(*
  :return: CamReady 
*)
METHOD GetCamStatus : BOOL
VAR_OUTPUT
  bConnectionOK  : BOOL;    // Camera connected
  bTeachOk       : BOOL;    // Teach successful
  nTeachedPoints : UDINT;   // Teached points for this job
  nScannedPoints : UDINT;   // Scanned points on current sheet  
  bCamStarted    : BOOL;    // Camera trigger is active, cam started
  bCamDone       : BOOL;    // Camera finished on CT
  bErrors        : ARRAY[1..GVL_Camera.nC_NbCamErrors] OF BOOL;  // generic error flag list
END_VAR
bConnectionOK  := NOT bConnectionErr OR bSimulate;
bTeachOk       := _bTeachOk OR bSimulate;
nTeachedPoints := nNbMarksTeach;
nScannedPoints := nNbMarksScanned;
bCamStarted    := _bCamTriggerStarted;
// camera finished
IF nNbVersion = cProtoVersion_110 THEN
  // Done: Trigger released and last sector was received
  bCamDone       := _bCamTriggerDone AND ((nSector >= nNbSectorTeach) OR (nSector = SINT_TO_DINT(-1)));
ELSE
  // Done: Trigger released and same all teached points are scanned // NOTE: this will not work if not all marks are detected by camera
  bCamDone       := _bCamTriggerDone AND (nScannedPoints>=nTeachedPoints);
END_IF
GetCamStatus := bConnectionOK AND bTeachOk;   // camera ready
END_METHOD

(*
  get array index to point ID in stored point table
  :returns: TRUE if found, FALSE else
*)
METHOD getPointIndex : BOOL
VAR_INPUT
  nId : UDINT;
END_VAR
VAR_OUTPUT
  nIndex : UDINT;
END_VAR
VAR
  nResultIdx : DINT;
END_VAR
// search corresponding point in table (search for same mark ID)

nResultIdx := binarySearch(1, TO_DINT(nNbMarksTeach), TO_DINT(nId));
IF nResultIdx = -1 THEN
  LogWarning(F_Concat3('Point with Id: ', TO_STRING(nId) , ' not found in saved teach points'));
  nIndex := 1;
  RETURN;
END_IF

nIndex := TO_UDINT(nResultIdx);
getPointIndex := TRUE;
END_METHOD

METHOD INTERNAL getSimCamPoint : ST_DeformationPointAccurate
VAR_INPUT
  fXMin : LREAL := 0.0;
	fXMax : LREAL := 0.0;
	fYMin : LREAL := 0.0;
	fYMax : LREAL := 0.0;
	
	fOffsetMin : LREAL := 0.0;
	fOffsetMax : LREAL := 0.0;
END_VAR
VAR_OUTPUT
  sO_CamPoint : ST_DeformationPointAccurate;
END_VAR
VAR_INST
  fbRand : DRAND;
END_VAR
fbRand();
sO_CamPoint.x_ref := (fXMin + (fXMax - fXMin));
fbRand();
sO_CamPoint.y_ref := (fYMin + (fYMax - fYMin));

fbRand();
sO_CamPoint.dx := (fOffsetMin + (fOffsetMax - fOffsetMin) * fbRand.Num);
fbRand();
sO_CamPoint.dy := (fOffsetMin + (fOffsetMax - fOffsetMin) * fbRand.Num);

sO_CamPoint.valid := _bSimCamPointValid;
getSimCamPoint := sO_CamPoint;
END_METHOD

METHOD InitLineCamera
VAR_INPUT
  nPrintUnitResolution         : UDINT;    (*printhead pixel resolution [dpi]*)
  nPrintUnitSubPx              : UDINT;    (*print unit subPixel resolution [SubPx]*)
  nPrintUnitWidth              : UDINT;    (*print unit width in [px]*)
  iCameraTrigger               : I_CameraTrigger;
END_VAR
_fCameraWidthNormal     := FC_CONV_SUBPX_TO_M( _nCameraWidth
                                             , LREAL_TO_UDINT(cCameraResolution)
                                             , 1);
_nPrintUnitWidthNormal  := nPrintUnitWidth;
_fPrintUnitCalTemp      := fC_PhPixelDistRefTemp;   // reference temperate for real pixel spacing of ph
_fPrintUnitWidthTC      := (nPrintUnitWidth * fC_PhPixelDistFactorAtRefTemp) / 1000;  // caluclate print unit with at calibration temperature [m]

SUPER^.Init( nPrintUnitResolution:=nPrintUnitResolution
           , nPrintUnitSubPx:=nPrintUnitSubPx
           , iCameraTrigger := iCameraTrigger
           , bUseCameraTrigger:=TRUE
           , bUseCameraTriggerFeedback:=TRUE);
END_METHOD

METHOD InitSimulation : BOOL
VAR_INPUT
  aCamSimScriptPath : T_MaxString;
END_VAR
_aCamSimScriptPath := aCamSimScriptPath;
END_METHOD

METHOD mJobStart : BOOL
// re-calculate teach points with previous received 'T' telegram 
//  handles case: teach telegram arrived before JobStart
IF sModus = 'T' THEN calcTeachPoints(); END_IF
END_METHOD

(*
  Tcpip client rx message callback. 
  Called by FB_TcpMsgNotifier, registered with 'registerTcpIpClient()' before.
*)
METHOD rx_callback
VAR_INPUT
  sMessage : CalmarCompTcpIp.ST_TcpMsg;    // rx message
END_VAR
VAR
  sAnalyzeLastMessage    : STRING(GVL_TcpIp.TCP_RXDATA_SIZE);          // telegram string for analysis
  sTmpCamPoint           : ST_CameraPoint;
  
  nCounter               : UDINT;
  bOk, bEnd              : BOOL;

END_VAR
// basic message handling
SUPER^.rx_callback(sMessage := sMessage);
// debug print
IF _bVerbose THEN LogLvl(Lvl:=E_LogSeverity.Debug,Msg:=F_Concat4('Rx Sz: ', TO_STRING(nLastMessageSz), ' Msg:', sLastMessage)); END_IF

// check parameter (avoids crash)
IF _fPrintUnitWidthTC = 0 THEN LogError('rx_callback: Invalid configuration, review persistences and config values!'); RETURN; END_IF

// copy for parsing
sAnalyzeLastMessage := sLastMessage;      

REPEAT
  (*--- check message type ---*)
  // -- Is it a test message?
  IF rx_TestMsg(pMessage:=ADR(sLastMessage)) THEN       (*Test message*)
    RETURN;   // test message, ignore rest of parsing
   
  // -- Is it a error message ?
  ELSIF rx_ErrorMsg(pMessage:=ADR(sLastMessage)) THEN   (*Error message*)
    RETURN;   // error message, ignore rest of parsing
  
  // -- Is it a position message ('T' Teach or 'A' Auswertung)
  ELSIF rx_ParseHeader( pAnalyzeLastMessage := ADR(sAnalyzeLastMessage)
                      , nNbVersion      => nNbVersion          (*version*)
                      , sModus          => sModus              (*modus*)
                      , nNbMarks        => nNbMarks            (*number of marks*)
                      , nSector         => nSector)            (*sector*)
    THEN
     // got a position message, do not exit and do rest of parsing below
     // >>> DO parsing below 
     ;
    
  // -- unknown message
  ELSE
    IF _bVerbose THEN LogLvl(Lvl:=E_LogSeverity.Debug, Msg:=F_Concat2('unknown rx message (ignore): ', sLastMessage)); END_IF
    RETURN;
  END_IF
  
  
  (*--- Handle position telegram ---*)
  IF (sModus  = 'T') THEN 
    (*-- 'T' Teach message *)
    nNbMarksTeach   := 0;
    nNbMarksScanned := 0;
    nNbSectorTeach  := nSector;  (*Total number or sectors are send with teach message.*)
    sTeach          := sAnalyzeLastMessage; // display on visu
    
    IF _bVerbose THEN LogLvl(Lvl:=E_LogSeverity.Debug, Msg:='receive T telegram, erase cam/teach points list'); END_IF    
    MEMSET(destAddr:=ADR(sTeachPoints),  fillByte:=0, n:=SIZEOF(sTeachPoints));   // eraase teach points list
    MEMSET(destAddr:=ADR(sCameraPoints), fillByte:=0, n:=SIZEOF(sCameraPoints));  // erase cam points list
    MEMSET(destAddr:=ADR(nNumPointsPerSectorA), fillByte:=0, n:=SIZEOF(nNumPointsPerSectorA));
    MEMSET(destAddr:=ADR(nNumPointsPerSectorT), fillByte:=0, n:=SIZEOF(nNumPointsPerSectorT));
  ELSE
    (*-- 'A' Auswertung message *)
    sMemLastMessage := sAnalyzeLastMessage; // display on visu
    
    IF nSector = TO_DINT(cIdxFirstSector) THEN  // erase campoint with first received sector
      MEMSET(destAddr:=ADR(sCameraPoints), fillByte:=0, n:=SIZEOF(sCameraPoints));  // erase cam points list
      IF _bVerbose THEN LogLvl(Lvl:=E_LogSeverity.Debug, Msg:=F_Concat2('received first A sector, erase cam points list.','')); END_IF
      
      _nTimeFrameIdx_CamMsg := 1;
    END_IF
  
    // debug timing rx A
    IF _nTimeFrameIdx_CamMsg <= nC_MaxRxTimingEntries THEN  // save message timestamp for debugging
      _tTimeFrames_CamMsg[_nTimeFrameIdx_CamMsg] := F_GetCurDcTaskTime64();     // save cam frame rx timestamp
      _tTimeFramesMs_CamMsg[_nTimeFrameIdx_CamMsg] := TO_LREAL((_tTimeFrames_CamMsg[_nTimeFrameIdx_CamMsg]-_tTimeTrigger)/EC_DCTIME_TICKSPERMSEC64);  // delta to trigger in ms
      IF _bVerbose THEN 
        // dbg log rx frames
        LogLvl(Lvl:=E_LogSeverity.Debug, Msg:=F_Concat4(
            F_Concat2('A-Frame: ', TO_STRING(_nTimeFrameIdx_CamMsg)),
            F_Concat2(' : ', TO_STRING(_nTimeFrameIdx_CamMsg)),
            F_Concat2(' after trig: ', TO_STRING(_tTimeFramesMs_CamMsg[_nTimeFrameIdx_CamMsg])),
            F_Concat2(' at: ', TO_STRING(_tTimeFrames_CamMsg[_nTimeFrameIdx_CamMsg]))
        ));
			END_IF
      _nTimeFrameIdx_CamMsg := _nTimeFrameIdx_CamMsg + 1;
    END_IF
    
  END_IF;
  
  
  (*Search for rx, ry, lx, ly, v, x and y*)
  FOR nCounter := 1 TO nNbMarks DO
    // get next point
    IF NOT rx_ParsePoint(pAnalyzeLastMessage:=ADR(sAnalyzeLastMessage), sCamResult=>sTmpCamPoint, bLast=>bEnd) THEN 
      // invalid point received
      LogWarning(F_Concat2(
        F_Concat3('invalid ', SEL(sModus='T', 'camera', 'teach'), ' point received, '),
        F_CamPoint_ToString(sPoint:=sTmpCamPoint)
      ));
    END_IF
    IF bEnd AND nCounter < nNbMarks THEN LogWarning(F_Concat4('Less marks received than indicated in header: ', TO_STRING(nCounter), '<', TO_STRING(nNbMarks))); END_IF
    
    IF (sModus  = 'T') THEN
      (*-- 'T' Teach message *)
      // save (convert with job start)
      saveTeachPoint(sCamPoint := sTmpCamPoint);
    ELSE
      (*-- 'A' Auswertung message *)
      // save & convert cam point
      stCamPoint := saveAuswertungPoint(sCamPoint:=sTmpCamPoint, bOK=>bOk);     
      // stream point (if valid)
      IF bOk THEN  //AND sTmpCamPoint.valid THEN
        IF _iCameraSink <> 0 THEN
          _iCameraSink.AddCamPoint(stCamPoint);
          IF _bVerbose THEN 
            LogLvl(Lvl:=E_LogSeverity.Debug, Msg:= F_Concat2('AddCamPoint: ', F_DeformationPointAcc_ToString(sPointAcc:=stCamPoint)));
          END_IF
        END_IF
      END_IF
    END_IF
  END_FOR
UNTIL FIND2(ADR(sAnalyzeLastMessage), ADR(cStartString)) = 0   (*Search for another start string*)
END_REPEAT

IF (sModus  = 'T') THEN calcTeachPoints(); END_IF  // calculate teach points if it was a teach

bMsgReceived := FALSE;
END_METHOD

METHOD PRIVATE rx_DeleteMsgPart
VAR_INPUT
  pAnalyzeLastMessage    : POINTER TO STRING(GVL_TcpIp.TCP_RXDATA_SIZE);  // telegram string for analysis
  nLen                   : UDINT;
  nPos                   : UDINT;
END_VAR
VAR
  sMessageDelete         : STRING(GVL_TcpIp.TCP_RXDATA_SIZE);             // telegram string for analysis
END_VAR
DELETE2( pSrcString := pAnalyzeLastMessage
       , pDstString := ADR(sMessageDelete)
       , nDstSize   := SIZEOF(sMessageDelete)
       , nLen       := nLen
       , nPos       := nPos);

pAnalyzeLastMessage^ := sMessageDelete;
END_METHOD

(*
  Parse for error message
  :return: TRUE if it was an error test telegram, FALSE if other.
*)
METHOD PRIVATE rx_ErrorMsg : BOOL
VAR_INPUT
  pMessage    : POINTER TO STRING(GVL_TcpIp.TCP_RXDATA_SIZE);   // tcp message string pointer 
END_VAR
VAR
  nFIdx : UDINT;    // string find index
  nFrmIdx : UDINT;
  tDiff : LREAL;
  sErrMsg : T_MaxString;
END_VAR
// parse message type
nFIdx := FIND2(pMessage, ADR(cErrorString));
IF nFIdx > 0 THEN  
  IF _bVerbose THEN LogLvl(Lvl:=E_LogSeverity.Debug, Msg:=F_Concat2('error: msg received: ', pMessage^)); END_IF

  // error telegram received
  DELETE2( pSrcString := pMessage
         , pDstString := ADR(sErrMsg)
         , nDstSize   := SIZEOF(sErrMsg)
         , nLen       := (nFIdx + INT_TO_UDINT(LEN(cErrorString)) - 1)
         , nPos       := 1);

  // strip other control characters
  FindAndDelete(pSrcString:=ADR(sErrMsg), pDstString:=ADR(sErrMsg), nDstSize:=SIZEOF(sErrMsg), pDeleteString:=ADR(cEndingString));
  
  // error message implement handling
  
  rx_ErrorMsg := TRUE;
ELSE
  ; // other telegram
END_IF
END_METHOD

(*
  Parse for position telegram header.
  :return: TRUE if valid position telegram, FALSE else
*)
METHOD PRIVATE rx_ParseHeader : BOOL
VAR_INPUT
  pAnalyzeLastMessage    : POINTER TO STRING(GVL_TcpIp.TCP_RXDATA_SIZE);  // telegram string for analysis
END_VAR
VAR_OUTPUT
  nNbVersion             : INT;                   (*(V) Version: protocol version, e.g. 100/110/...*)
  sModus                 : T_MaxString;           (*(M) Modus: 'T'/'A'*)
  nNbMarks               : UDINT;                 (*(A) Merkmale: number of Marks in Teach/Auswertung*)
  nSector                : DINT;                  (*(S) Sectors: Number of Sectors in 'T' / Sector index in 'A'*)
  //sMemLastMessage        : STRING(GVL_TcpIp.TCP_RXDATA_SIZE);  (*rx telegram string without header*)
END_VAR
VAR
  nFindIndex             : UDINT;
END_VAR
(*Search for start string*)
nFindIndex := FIND2(pAnalyzeLastMessage, ADR(cStartString));
IF nFindIndex = 0 THEN RETURN; END_IF

(*Search string found => remove string to evaluate rest of message*)
rx_DeleteMsgPart(pAnalyzeLastMessage := pAnalyzeLastMessage, nLen := (nFindIndex + INT_TO_UDINT(LEN(cStartString)) - 1) , nPos := 1);

(*Search for version number*)
nFindIndex := FIND2(pAnalyzeLastMessage, ADR(','));
IF nFindIndex > 0 THEN
  nNbVersion := STRING_TO_INT(LEFT(pAnalyzeLastMessage^, (UDINT_TO_INT(nFindIndex) - 1)));

  rx_DeleteMsgPart(pAnalyzeLastMessage := pAnalyzeLastMessage, nLen := nFindIndex , nPos := 1);
END_IF;

(*Search for modus (M)*)
nFindIndex := FIND2(pAnalyzeLastMessage, ADR(','));
IF nFindIndex > 0 THEN
  sModus := LEFT(pAnalyzeLastMessage^, (UDINT_TO_INT(nFindIndex) - 1));

  rx_DeleteMsgPart(pAnalyzeLastMessage := pAnalyzeLastMessage, nLen := nFindIndex , nPos := 1);
END_IF;

(*Search for number marks (A)*)
nFindIndex := FIND2(pAnalyzeLastMessage, ADR(','));
IF nFindIndex > 0 THEN
  nNbMarks := STRING_TO_UDINT(LEFT(pAnalyzeLastMessage^, (UDINT_TO_INT(nFindIndex) - 1)));
  IF nNbMarks > GVL_Camera.cMaxNbMarks THEN
    LogLvl(Lvl:=E_LogSeverity.Warning, Msg:=F_Concat4('Limit marks (', TO_STRING(nNbMarks),') to max=', TO_STRING(GVL_Camera.cMaxNbMarks)));
    nNbMarks := GVL_Camera.cMaxNbMarks;
  END_IF

  rx_DeleteMsgPart(pAnalyzeLastMessage := pAnalyzeLastMessage, nLen := nFindIndex , nPos := 1);
END_IF;

(*Search for sector of transmission (S)*)
nFindIndex := FIND2(pAnalyzeLastMessage, ADR(','));
IF nFindIndex > 0 THEN
  (*Last sector is indicated with '-1'*)
  nSector := STRING_TO_DINT(LEFT(pAnalyzeLastMessage^, (UDINT_TO_INT(nFindIndex) - 1)));

  rx_DeleteMsgPart(pAnalyzeLastMessage := pAnalyzeLastMessage, nLen := nFindIndex , nPos := 1);
ELSE
  // end of message detected
  nFindIndex := FIND2(pAnalyzeLastMessage, ADR(');'));
  IF nFindIndex > 0 THEN
    (*Last sector is indicated with '-1'*)
    nSector := STRING_TO_DINT(LEFT(pAnalyzeLastMessage^, (UDINT_TO_INT(nFindIndex) - 1)));
  
    rx_DeleteMsgPart(pAnalyzeLastMessage := pAnalyzeLastMessage, nLen := nFindIndex + 1, nPos := 1);
  END_IF;
END_IF;

rx_ParseHeader := TRUE;
END_METHOD

(*
  Parse a point entry from string.
  And removes this string part from pAnalyzeLastMessage.
  :return: TRUE if point is valid
*)
METHOD PRIVATE rx_ParsePoint : BOOL
VAR_INPUT
  pAnalyzeLastMessage    : POINTER TO STRING(GVL_TcpIp.TCP_RXDATA_SIZE);  // telegram string for analysis
END_VAR
VAR_OUTPUT
  sCamResult             : ST_CameraPoint;
  bLast                  : BOOL;
END_VAR
VAR
  nFindIndex             : UDINT;
END_VAR
(*Index of mark (T)*)
nFindIndex := FIND2(pAnalyzeLastMessage, ADR(','));
IF nFindIndex > 0 THEN
  sCamResult.id := STRING_TO_UDINT(LEFT(pAnalyzeLastMessage^, (UDINT_TO_INT(nFindIndex) - 1)));
  
  rx_DeleteMsgPart(pAnalyzeLastMessage := pAnalyzeLastMessage, nLen := nFindIndex , nPos := 1);
END_IF;

(*rx*)
nFindIndex := FIND2(pAnalyzeLastMessage, ADR(','));
IF nFindIndex > 0 THEN
  sCamResult.x_ref := STRING_TO_DINT(LEFT(pAnalyzeLastMessage^, (UDINT_TO_INT(nFindIndex) - 1)));

  IF    (sCamResult.x_ref < cCameraMinXY)
     OR (sCamResult.x_ref > cCameraMaxXY)
  THEN
    sCamResult.valid := FALSE;
  END_IF;

  rx_DeleteMsgPart(pAnalyzeLastMessage := pAnalyzeLastMessage, nLen := nFindIndex , nPos := 1);
ELSE
  sCamResult.valid := FALSE;
END_IF;
(*ry*)
nFindIndex := FIND2(pAnalyzeLastMessage, ADR(','));
IF nFindIndex > 0 THEN
  sCamResult.y_ref := STRING_TO_DINT(LEFT(pAnalyzeLastMessage^, (UDINT_TO_INT(nFindIndex) - 1)));

  IF    (sCamResult.y_ref < cCameraMinXY)
     OR (sCamResult.y_ref > cCameraMaxXY)
  THEN
    sCamResult.valid := FALSE;
  END_IF;

  rx_DeleteMsgPart(pAnalyzeLastMessage := pAnalyzeLastMessage, nLen := nFindIndex , nPos := 1);
ELSE
  sCamResult.valid := FALSE;
END_IF;

(*lx*)
nFindIndex := FIND2(pAnalyzeLastMessage, ADR(','));
IF nFindIndex > 0 THEN
  sCamResult.lx := STRING_TO_DINT(LEFT(pAnalyzeLastMessage^, (UDINT_TO_INT(nFindIndex) - 1)));

  IF    (sCamResult.lx < cCameraMinXY)
     OR (sCamResult.lx > cCameraMaxXY)
  THEN
    sCamResult.valid := FALSE;
  END_IF;

  rx_DeleteMsgPart(pAnalyzeLastMessage := pAnalyzeLastMessage, nLen := nFindIndex , nPos := 1);
ELSE
  sCamResult.valid := FALSE;
END_IF;
(*ly*)
nFindIndex := FIND2(pAnalyzeLastMessage, ADR(','));
IF nFindIndex > 0 THEN
  sCamResult.ly := STRING_TO_DINT(LEFT(pAnalyzeLastMessage^, (UDINT_TO_INT(nFindIndex) - 1)));

  IF    (sCamResult.ly < cCameraMinXY)
     OR (sCamResult.ly > cCameraMaxXY)
  THEN
    sCamResult.valid := FALSE;
  END_IF;

  rx_DeleteMsgPart(pAnalyzeLastMessage := pAnalyzeLastMessage, nLen := nFindIndex , nPos := 1);
ELSE
  sCamResult.valid := FALSE;
END_IF;

(*v*)
nFindIndex := FIND2(pAnalyzeLastMessage, ADR(','));
IF nFindIndex > 0 THEN
  IF STRING_TO_INT(LEFT(pAnalyzeLastMessage^, (UDINT_TO_INT(nFindIndex) - 1))) = 1 THEN
    sCamResult.valid := TRUE;
  ELSE
    sCamResult.valid := FALSE;
  END_IF;

  rx_DeleteMsgPart(pAnalyzeLastMessage := pAnalyzeLastMessage, nLen := nFindIndex , nPos := 1);
ELSE
  sCamResult.valid := FALSE;
END_IF;
(*x*)
nFindIndex := FIND2(pAnalyzeLastMessage, ADR(','));
IF nFindIndex > 0 THEN
  sCamResult.x := STRING_TO_DINT(LEFT(pAnalyzeLastMessage^, (UDINT_TO_INT(nFindIndex) - 1)));

  IF    (sCamResult.x < cCameraMinXY)
     OR (sCamResult.x > cCameraMaxXY)
  THEN
    sCamResult.valid := FALSE;
  END_IF;

  rx_DeleteMsgPart(pAnalyzeLastMessage := pAnalyzeLastMessage, nLen := nFindIndex , nPos := 1);
ELSE
  sCamResult.valid := FALSE;
END_IF;
(*y*)
nFindIndex := FIND2(pAnalyzeLastMessage, ADR(','));
IF (nFindIndex > 0) AND (nFindIndex <= 8) THEN  (*nFindIndex is > 8 if a second message is in the frame*)
  sCamResult.y := STRING_TO_DINT(LEFT(pAnalyzeLastMessage^, (UDINT_TO_INT(nFindIndex) - 1)));

  IF    (sCamResult.y < cCameraMinXY)
     OR (sCamResult.y > cCameraMaxXY)
  THEN
    sCamResult.valid := FALSE;
  END_IF;

  rx_DeleteMsgPart(pAnalyzeLastMessage := pAnalyzeLastMessage, nLen := nFindIndex , nPos := 1);
ELSE
  nFindIndex := FIND2(pAnalyzeLastMessage, ADR(');'));
  IF nFindIndex > 0 THEN
    sCamResult.y := STRING_TO_DINT(LEFT(pAnalyzeLastMessage^, (UDINT_TO_INT(nFindIndex) - 1)));
    bLast := TRUE;
    IF    (sCamResult.y < cCameraMinXY)
       OR (sCamResult.y > cCameraMaxXY)
    THEN
      sCamResult.valid := FALSE;
    END_IF;

    rx_DeleteMsgPart(pAnalyzeLastMessage := pAnalyzeLastMessage, nLen := nFindIndex + 1, nPos := 1);
  ELSE
    sCamResult.valid := FALSE;
  END_IF;
END_IF;

rx_ParsePoint := sCamResult.valid;
END_METHOD

(*
  Parse rx test telegrams.
  :return: TRUE if it was a known test telegram, FALSE if other.
*)
METHOD PRIVATE rx_TestMsg : BOOL
VAR_INPUT
  pMessage    : POINTER TO STRING(GVL_TcpIp.TCP_RXDATA_SIZE);   // tcp message string pointer 
END_VAR
VAR
  nFIdx : UDINT;    // string find index
  nFrmIdx : UDINT;
  tDiff : LREAL;
  sTestMsg : T_MaxString;
END_VAR
// rx timestamp
_tTimeRx := F_GetCurDcTaskTime64();

// parse message type
nFIdx := FIND2(pMessage, ADR(sQvTest_Header));
IF nFIdx > 0 THEN  
  IF _bVerbose THEN
    LogLvl(Lvl:=E_LogSeverity.Debug, Msg:=F_Concat2('test_rx: msg received: ', pMessage^));
  END_IF
  
  // test telegram received
  DELETE2( pSrcString := pMessage
         , pDstString := ADR(sTestMsg)
         , nDstSize   := SIZEOF(sTestMsg)
         , nLen       := (nFIdx + INT_TO_UDINT(LEN(sQvTest_Header)) - 1)
         , nPos       := 1);

  // strip QR start and end characters
  FindAndDeleteChar(pSrcString:=ADR(sTestMsg), pDstString:=ADR(sTestMsg), nDstSize:=SIZEOF(sTestMsg), sDeleteChar:='<');
  FindAndDeleteChar(pSrcString:=ADR(sTestMsg), pDstString:=ADR(sTestMsg), nDstSize:=SIZEOF(sTestMsg), sDeleteChar:=';');
  
  // Parse per test message type, e.g.  <QR_CI_1;
  // -- qv input frame timing test
  IF sQvTest_CI = LEFT(sTestMsg, LEN(sQvTest_CI)) THEN
    // strip header and test indication
    DELETE2( pSrcString := ADR(sTestMsg)
           , pDstString := ADR(sTestMsg)
           , nDstSize   := SIZEOF(sTestMsg)
           , nLen       := (1 + INT_TO_UDINT(LEN(sQvTest_CI)) - 1)
           , nPos       := 1);
    // frame number
    nFrmIdx := TO_UINT(sTestMsg);
    IF nFrmIdx <= nC_MaxRxTimingEntries THEN
      _tTimeFrames_TestMsg[nFrmIdx] := F_GetCurDcTaskTime64();     // save test input frame timestamp
      _tTimeFramesMs_TestMsg[nFrmIdx] := TO_LREAL((_tTimeFrames_TestMsg[nFrmIdx]-_tTimeTrigger)/EC_DCTIME_TICKSPERMSEC64);
    END_IF
    rx_TestMsg := TRUE;
    
  // -- qv loop time test frame response
  ELSIF sQvTest_Loop = LEFT(sTestMsg, LEN(sQvTest_Loop)) THEN
    tDiff := TO_LREAL((_tTimeRx - _tTimeTx) / EC_DCTIME_TICKSPERMSEC64); // calc time elapsed in [ms]
    _sTimeElapsed := F_Concat2(TO_STRING(tDiff),'ms');
    LogLvl(Lvl:=E_LogSeverity.Debug, Msg:=F_Concat2('rx_test: Loop time=', _sTimeElapsed));
    rx_TestMsg := TRUE;
  
  // -- unknown test message
  ELSE
    ;
	END_IF
ELSE
  ; // other telegram
END_IF
END_METHOD

METHOD PRIVATE saveAuswertungPoint : ST_DeformationPointAccurate
VAR_INPUT
  sCamPoint : ST_CameraPoint;
END_VAR
VAR_OUTPUT
  bOK : BOOL;   // conversion has been done correctly (ok as well if point is invalid!)
END_VAR
VAR
  nMarkIndex        : UDINT;
  fDistortionFactor : LREAL;                 (*distortion factor*)
END_VAR
(*convert and save Auswertungs point*)
IF NOT getPointIndex(nId:=sCamPoint.id, nIndex=>nMarkIndex) THEN
  LogError(F_Concat3('Auswertung point with Id: ', TO_STRING(sCamPoint.id), ' not found, ignore'));
  bOK := FALSE;
  RETURN;
END_IF

(*----- calculate print point position -----*)
(*Actual position of distinctive mark*)
(*NOTE: camera points have a different resolution! camera 300dpi * 16=4800dpi*)
IF sTeachPoints[nMarkIndex].x_teach_Print = 0 THEN 
  (*Fully automatic mode*)
  sTeachPoints[nMarkIndex].x_Print := FC_CONV_SUBPX_TO_M( sCamPoint.y
                                                          , LREAL_TO_UDINT(cCameraResolution)
                                                          , LREAL_TO_UDINT(cCameraResolutionSubpixel)) * 1000;  (*[m] => [mm]*)
ELSE
  (*Semi automatic mode*)
  sTeachPoints[nMarkIndex].x_Print :=     sTeachPoints[nMarkIndex].x_ref_Print
                                        + sTeachPoints[nMarkIndex].x_teach_Print
                                        - FC_CONV_SUBPX_TO_M( sCamPoint.y
                                                            , LREAL_TO_UDINT(cCameraResolution)
                                                            , LREAL_TO_UDINT(cCameraResolutionSubpixel)) * 1000;  (*[m] => [mm]*)
END_IF;
IF sTeachPoints[nMarkIndex].y_teach_Print = 0 THEN 
  (*Fully automatic mode*)
  sTeachPoints[nMarkIndex].y_Print :=   ((fPrintUnitWidthTAct/2 + fCameraWidthTC/2) * 1000)  (*[m] => [mm]*)
                                        - (  DINT_TO_LREAL(sCamPoint.x)
                                           / (fCameraRealResolution * cCameraResolutionSubpixel) * 25.4);  (*[mm]*)
ELSE
  (*Semi automatic mode*)
  sTeachPoints[nMarkIndex].y_Print :=     sTeachPoints[nMarkIndex].y_ref_Print
                                        + sTeachPoints[nMarkIndex].y_teach_Print
                                        - (  DINT_TO_LREAL(sCamPoint.x)
                                           / (fCameraRealResolution * cCameraResolutionSubpixel) * 25.4);  (*[mm]*)
END_IF;

// save cam point for visu
sCameraPoints[nMarkIndex] := sCamPoint;

(*----- create cam correction point -----*)
(*NOTE: correction will be rounded to [px]*)
saveAuswertungPoint.x_ref := F_MeterToSubPixelReal( sTeachPoints[nMarkIndex].x_ref_Print * 0.001      (*[mm] => [m]*)
                                     , UDINT_TO_LREAL(_nPrintUnitResolution));             (*Result should be in pixels*)                           
saveAuswertungPoint.y_ref := F_MeterToSubPixelReal( sTeachPoints[nMarkIndex].y_ref_Print * 0.001      (*[mm] => [m]*)
                                     , UDINT_TO_LREAL(_nPrintUnitResolution));             (*Result should be in pixels*)       
fCameraDelay := F_SubPixelToMeter(lPosSubPx:=_nCamStartPosDeviation, fResSubPx:=UDINT_TO_LREAL(_nPrintUnitResolution*_nPrintUnitSubPx));
saveAuswertungPoint.dx    := F_MeterToSubPixelReal( (sTeachPoints[nMarkIndex].x_ref_Print - sTeachPoints[nMarkIndex].x_Print) * 0.001  (*[mm] => [m]*)
                                     + fCameraDelay                                        (*apply camera trigger jitter*)
                                     , UDINT_TO_LREAL(_nPrintUnitResolution));             (*Result should be in pixels*)
                                     
(*Distortion due to expansion of print unit, calculate factor*)
fDistortionFactor := ((_fPrintUnitWidthTC / 2 * 1000) - sTeachPoints[nMarkIndex].y_ref_Print) / (_fPrintUnitWidthTC / 2 * 1000);
saveAuswertungPoint.dy := F_MeterToSubPixelReal( (  (sTeachPoints[nMarkIndex].y_ref_Print - sTeachPoints[nMarkIndex].y_Print)
                                     + fCameraAdjustmentY
                                     + ((fPrintUnitWidthDiff * 1000 / 2) * fDistortionFactor)   (*Distortion due to expansion of print unit*)
                                     + (fPrintUnitCenterOffsetTAct - fCameraCenterOffsetTAct)   (*Compensation due to unilateral expansion*)
                                    ) * 0.001  (*[mm] => [m]*)
                                  , UDINT_TO_LREAL(_nPrintUnitResolution));             (*Result should be in pixels*)
                                  
// not used entries
saveAuswertungPoint.index := 0; // optional: TO_DINT(sCamPoint.id);
saveAuswertungPoint.col := 0;
saveAuswertungPoint.row := 0;
saveAuswertungPoint.valid := sCamPoint.valid;
IF NOT sCamPoint.valid THEN     // erase spurious corrections on invalid points
  saveAuswertungPoint.dx := 0;
  saveAuswertungPoint.dy := 0;
END_IF
nNbMarksScanned := nNbMarksScanned + 1;
bOK := TRUE;
END_METHOD

METHOD PRIVATE saveTeachPoint
VAR_INPUT
  sCamPoint : ST_CameraPoint;
END_VAR
(*save teach point in table*)
// NOTE: mark ID unique and does not match the array index! 
IF nNbMarksTeach = GVL_Camera.cMaxNbMarks THEN 
  LogLvl(Lvl:=E_LogSeverity.Error, Msg:=F_Concat4('Too many marks received max. allowed: ', TO_STRING(GVL_Camera.cMaxNbMarks), ' ignore mark with id:', TO_STRING(sCamPoint.id)));
  RETURN;
END_IF

// save next teach mark
nNbMarksTeach := nNbMarksTeach + 1;
sCameraPoints[nNbMarksTeach] := sCamPoint;
END_METHOD

(*
  Set mode to camera.
  :return: TRUE if success
*)
METHOD setCameraMode : BOOL
VAR_INPUT
  eCameraMode : E_CameraMode;
END_VAR
IF eCameraMode = E_CameraMode.XYR OR   // supported modi
   eCameraMode = E_CameraMode.Auto OR
   eCameraMode = E_CameraMode.Live OR 
   eCameraMode = E_CameraMode.Trend THEN
   
  _eCameraMode := eCameraMode;  // set desired mode
  setCameraMode := TRUE;
ELSE
  LogError(F_Concat3('Camera mode=', TO_STRING(eCameraMode), ' not supported by camera'));
  _eCameraMode := E_CameraMode.NoCorrection;
END_IF
END_METHOD

METHOD SimEnter : BOOL
VAR_INST
  sSimMsg         : CalmarCompTcpIp.ST_TcpMsg;
  nFrameSize      : UDINT := 2048;
  nMarksPerFrame  : UDINT := 4;
END_VAR
IF NOT bSimEnable THEN RETURN; END_IF

IF    _nSimMode = 0 THEN
   //nNbMarksTeach := 4; // just somebigger than 2
   //nNbMarks := nNbMarksTeach;
ELSIF _nSimMode = 1 THEN
  // use external camera simulation script
  nFrameNr := 0;
ELSIF _nSimMode = 2 THEN
  // send directly some messages
  sSimMsg.stRemoteAddr.sAddr:='127.0.0.1';
  sSimMsg.stRemoteAddr.nPort:=3000;
  //v100 teach
  //rx_callback(sMessage:='<position(100,T,39,3,125,0,0,0,0,1,7184,7184,126,0,0,0,0,1,7184,26080,127,0,0,0,0,1,7184,35520,128,0,0,0,0,1,7184,54416,129,0,0,0,0,1,7168,73312,130,0,0,0,0,1,7184,82768,131,0,0,0,0,1,7184,101664,132,0,0,0,0,1,7184,120560,133,0,0,0,0,1,7184,139456,134,0,0,0,0,1,7184,148912,135,0,0,0,0,1,7184,167808,136,0,0,0,0,1,7168,186704,137,0,0,0,0,1,63872,7184,138,0,0,0,0,1,63872,26080,139,0,0,0,0,1,63872,35520,140,0,0,0,0,1,63872,54416,141,0,0,0,0,1,63872,73312,142,0,0,0,0,1,63872,82768,143,0,0,0,0,1,63872,101664,144,0,0,0,0,1,63872,120560,145,0,0,0,0,1,63872,139456,146,0,0,0,0,1,63872,148912,147,0,0,0,0,1,63872,167808,148,0,0,0,0,1,63872,186704,149,0,0,0,0,1,130016,7168,150,0,0,0,0,1,130016,26080,151,0,0,0,0,1,130016,35520,152,0,0,0,0,1,130016,54416,153,0,0,0,0,1,130016,73312,154,0,0,0,0,1,130016,82768,155,0,0,0,0,1,130016,101664,156,0,0,0,0,1,130016,120560,157,0,0,0,0,1,130016,139456,158,0,0,0,0,1,130016,148912,159,0,0,0,0,1,130016,167808,160,0,0,0,0,1,130016,186704,161,0,0,0,0,1,35520,7168,162,0,0,0,0,1,35520,5441);');
  //v110 teach
  sSimMsg.sMessage:= '<position(110,T,38,12,1,0,0,0,0,1,7184,7184,2,0,0,0,0,1,7184,26080,4,0,0,0,0,1,7184,35520,128,0,0,0,0,1,7184,54416,5,0,0,0,0,1,7168,73312,130,0,0,0,0,1,7184,82768,131,0,0,0,0,1,7184,101664,132,0,0,0,0,1,7184,120560,133,0,0,0,0,1,7184,139456,134,0,0,0,0,1,7184,148912,135,0,0,0,0,1,7184,167808,136,0,0,0,0,1,7168,186704,137,0,0,0,0,1,63872,7184,138,0,0,0,0,1,63872,26080,139,0,0,0,0,1,63872,35520,140,0,0,0,0,1,63872,54416,141,0,0,0,0,1,63872,73312,142,0,0,0,0,1,63872,82768,143,0,0,0,0,1,63872,101664,144,0,0,0,0,1,63872,120560,145,0,0,0,0,1,63872,139456,146,0,0,0,0,1,63872,148912,147,0,0,0,0,1,63872,167808,148,0,0,0,0,1,63872,186704,149,0,0,0,0,1,130016,7168,150,0,0,0,0,1,130016,26080,151,0,0,0,0,1,130016,35520,152,0,0,0,0,1,130016,54416,153,0,0,0,0,1,130016,73312,154,0,0,0,0,1,130016,82768,155,0,0,0,0,1,130016,101664,156,0,0,0,0,1,130016,120560,157,0,0,0,0,1,130016,139456,158,0,0,0,0,1,130016,148912,159,0,0,0,0,1,130016,167808,160,0,0,0,0,1,130016,186704,161,0,0,0,0,1,35520,7168,162,0,0,0,0,1,35520,5441);';
  //points 1 to 38
  //sSimMsg.sMessage:= '<position(110,T,38,12,1,0,0,0,0,1,7184,7184,2,0,0,0,0,1,7184,26080,3,0,0,0,0,1,7184,35520,4,0,0,0,0,1,7184,54416,5,0,0,0,0,1,7168,73312,6,0,0,0,0,1,7184,82768,7,0,0,0,0,1,7184,101664,8,0,0,0,0,1,7184,120560,9,0,0,0,0,1,7184,139456,10,0,0,0,0,1,7184,148912,11,0,0,0,0,1,7184,167808,12,0,0,0,0,1,7168,186704,13,0,0,0,0,1,63872,7184,14,0,0,0,0,1,63872,26080,15,0,0,0,0,1,63872,35520,16,0,0,0,0,1,63872,54416,17,0,0,0,0,1,63872,73312,18,0,0,0,0,1,63872,82768,19,0,0,0,0,1,63872,101664,20,0,0,0,0,1,63872,120560,21,0,0,0,0,1,63872,139456,22,0,0,0,0,1,63872,148912,23,0,0,0,0,1,63872,167808,24,0,0,0,0,1,63872,186704,25,0,0,0,0,1,130016,7168,26,0,0,0,0,1,130016,26080,27,0,0,0,0,1,130016,35520,28,0,0,0,0,1,130016,54416,29,0,0,0,0,1,130016,73312,30,0,0,0,0,1,130016,82768,31,0,0,0,0,1,130016,101664,32,0,0,0,0,1,130016,120560,33,0,0,0,0,1,130016,139456,34,0,0,0,0,1,130016,148912,35,0,0,0,0,1,130016,167808,36,0,0,0,0,1,130016,186704,37,0,0,0,0,1,35520,7168,38,0,0,0,0,1,35520,5441);';
  rx_callback(sMessage:=sSimMsg);
END_IF
END_METHOD

METHOD SimExit : BOOL
IF NOT bSimEnable THEN RETURN; END_IF

IF    _nSimMode = 0 THEN
  ;  // no action
ELSIF _nSimMode = 1 THEN
  nFrameNr := 0;
ELSIF _nSimMode = 2 THEN
  ;  // no action
END_IF
END_METHOD

(*
  External camera simulation script. 
  Simulates the line camera. Opens a TcpIp server where the the linecam plc client can conect to...
*)
METHOD SimulateCamera
VAR_INST
  rfTrig_En : RF_TRIG;
  tOnFrame  : TON;
END_VAR
VAR
  ams_host : STRING;
  ams_port : UINT;
  cmd : STRING;
  
  tFrameTime : TIME;
END_VAR
IF _nSimMode <> 1 THEN RETURN; END_IF   // only cam simulation

// simulation enable / disable
rfTrig_En(CLK:=_bSimulate);
IF rfTrig_En.RT THEN 
  // --- start simulation -----
  LogLvl(Lvl:=E_LogSeverity.Debug, Msg:='Start CamSimulation');

  fbScriptCamSim.Init(sScriptDir:=F_Concat2(_aCamSimScriptPath, 'Tools\CameraTest\'));
  fbScriptCamSim.sStartScriptName := 'Start.bat';
  (* Script parameter:
    parser.add_argument("ams_host", help="AmsNetId of host system")
    parser.add_argument("ams_port", help="AmsPort of host system", type=int)
    parser.add_argument("plc_path", help="plc interface (base) path")
    parser.add_argument("cam_ip", help="camera ip address")
    parser.add_argument("cam_port", help="camera port")
    parser.add_argument("--sim_mode", help="simulation enabled", type=bool)
  *)
  // build cmd line string dynamically 
  ams_host := '';
  ams_port := TwinCAT_SystemInfoVarList._AppInfo.AdsPort; 
  cmd := F_Concat7(ams_host,' ',TO_STRING(ams_port),' ',THIS^.InstanceName,' ',F_Concat3('127.0.0.1',' ',TO_STRING(5030)));
  fbScriptCamSim.Start(cmd);
  
ELSIF rfTrig_En.FT THEN 
  // --- stop/exit simulation ------
  LogLvl(Lvl:=E_LogSeverity.Debug, Msg:='Stop CamSimulation');
  // stop script
  fbScriptCamSim.Stop(nPID := THIS^.nScriptPID);
END_IF

// --- run script command ------
IF NOT fbScriptCamSim.bBusy THEN 
  IF fbScriptCamSim.bError THEN //Launch error
    LogError(F_Concat2('Script error=', TO_STRING(fbScriptCamSim.nErrId)));
  ELSE //Launch done
    ;
  END_IF
END_IF

// --- script live interface -------
IF _bCamTriggerStarted THEN
  IF tOnFrame.Q THEN
    nFrameNr := nFrameNr + 1; // demand next frame
	END_IF
  tFrameTime := REAL_TO_TIME(((84.6667 / 1_000_000) * 0.5)*1000*1024);  // 1024px @300dpi with speed 0.5m/s
  tOnFrame(IN:=NOT tOnFrame.Q, PT:=tFrameTime);
END_IF
END_METHOD

METHOD SimUpdate : BOOL
VAR_INST
  rfTrigCamTrigger : RF_TRIG;
  sSimMsg          : CalmarCompTcpIp.ST_TcpMsg;
END_VAR
// simulation handling
_rfTrigSim(CLK:=_bSimulate);
IF _rfTrigSim.RT THEN    SimEnter();
ELSIF _rfTrigSim.FT THEN SimExit(); END_IF
IF NOT _bSimulate THEN RETURN; END_IF

// we are in simulation mode
// - triggered
rfTrigCamTrigger(CLK:=_bCamTriggerStarted);

IF    _nSimMode = 0 THEN
  // direct points stream of all points in trigger
  IF rfTrigCamTrigger.RT THEN
     CreateSimCamPoints();
     _ePossibleMode := E_CameraMode.Live;
  END_IF
  // stream points
  StreamSimCamPoint();
 
ELSIF _nSimMode = 1 THEN
  // use external camera simulation script
  SimulateCamera();
  
ELSIF _nSimMode = 2 THEN
  IF rfTrigCamTrigger.RT THEN
    // send directly some messages
    sSimMsg.sMessage:='<position(110,A,5,1,125,0,0,0,0,1,12196,9766,137,0,0,0,0,1,69013,9660,149,0,0,0,0,1,135374,9496,161,0,0,0,0,1,40589,9699,163,0,0,0,0,1,116414,9527);';
    rx_callback(sMessage:=sSimMsg);
    sSimMsg.sMessage:='<position(110,A,3,2,126,0,0,0,0,1,11602,28300,138,0,0,0,0,1,68917,28190,150,0,0,0,0,1,136214,27951);';
    // also posible: sSimMsg.sMessage:='<position(110,A,3,2,126,0,0,0,0,1,11602,28300,138,0,0,0,0,1,68917,28190,150,0,0,0,0,1,136214,27951);<position(110,A,0,-1);';
    rx_callback(sMessage:=sSimMsg);
    sSimMsg.sMessage:='<position(110,A,0,-1);';
    rx_callback(sMessage:=sSimMsg);
  END_IF
END_IF


tx_test();
END_METHOD

{attribute 'monitoring':='variable'}
PROPERTY sName : STRING
GET
sName := 'LineCam Base';
END_GET
END_PROPERTY

(*
  Sort sCameraPoints list with ascending [.id] 
*)
METHOD sortPoints
VAR
  i, k : UDINT;
  tmpPoint : ST_CameraPoint;
END_VAR
// sort array (increasing id)
FOR i := 1 TO nNbMarksTeach DO
  FOR k := 1 TO nNbMarksTeach-1 DO
    IF sCameraPoints[k].id > sCameraPoints[k+1].id THEN
      tmpPoint := sCameraPoints[k+1];
      sCameraPoints[k+1] := sCameraPoints[k];
      sCameraPoints[k] := tmpPoint;
    END_IF
	END_FOR
END_FOR
END_METHOD

METHOD PRIVATE StreamSimCamPoint : BOOL
VAR_INPUT
END_VAR
VAR
 tCurrent : T_DCTIME64;
 tElapsed : LREAL;
 tCol : LREAL;
 nCol : UDINT;
 nPointCt : UDINT;
 tFrameFirstDelayFix : LREAL := 50; // deleat to first received frame after trigger
 tFrameTimeJitterMax : LREAL := 30; // max. process time for a camera frame to be received after a simulated scan [ms]
END_VAR
VAR_INST
 fbRand : DRAND;
END_VAR
IF IfSpeed = 0 THEN RETURN; END_IF

fbRand();
tCurrent := F_GetCurDcTaskTime64();             // current time 
tElapsed := TO_LREAL((tCurrent-_tTimeTrigger)   // time elapsed after trigger
                  / EC_DCTIME_TICKSPERMSEC64); 
tCol := F_SubPixelToMeter(                      // time for one column  in [ms] 
                  lPosSubPx:=TO_DINT(_nSimCamFrameDepth), 
                  fResSubPx:=_nPrintUnitResolution) * 1000 / IfSpeed;
tElapsed := tElapsed-tFrameFirstDelayFix-(tFrameTimeJitterMax * fbRand.Num);
IF tElapsed < 0 THEN nCol := 0;
ELSE                 nCol := TO_UDINT(tElapsed / tCol);  // current column number
END_IF

nPointCt := nCol*_nSimCamMarksPerFrame;         // current number of points to be streamed

// stream new points
WHILE nNbMarksScanned < nPointCt AND nNbMarksScanned < nNbMarks DO
  // add to container
  IF _iCameraSink<>0 THEN
    stCamPoint := _sSimCamPoints[nNbMarksScanned+1];
    _iCameraSink.AddCamPoint(stCamPoint);
    // add scanned marks
  END_IF;
  nNbMarksScanned := nNbMarksScanned + 1;
END_WHILE
END_METHOD

METHOD PRIVATE tx_test : BOOL
VAR_INPUT
END_VAR
VAR_INST
  _sTestTxMsg               : T_MaxString;
END_VAR
IF _pFbTcpIpClient = 0 THEN RETURN; END_IF

// sent a test message to QR
IF _bTestTx THEN
  _sTestTxMsg := F_Concat4('<', sQvTest_Header, sQvTest_Loop, ';');
  _tTimeTx := F_GetCurDcTaskTime64();
  _pFbTcpIpClient^.send(sMessage:=_sTestTxMsg);
  LogLvl(Lvl:=E_LogSeverity.Debug, Msg:=F_Concat2('test_tx sent: ', _sTestTxMsg));
  _bTestTx := FALSE;
END_IF
END_METHOD

(*
  Check teach points for validy and quality.
*)
METHOD verifyTeachPoints : BOOL
VAR
  lCtr : UDINT;
END_VAR

IF _fFrameLength <> 0 THEN
  nNumFrames := LIMIT(1, TO_UDINT(FC_LREAL_TO_DINT((fImageLength / _fFrameLength) + 1)), GVL_Camera.cMaxNbSectors); 
END_IF
bNotAllFramesContainTeachPoints := FALSE;
FOR lCtr := 1 TO nNumFrames DO
  IF nNumPointsPerSectorT[lCtr] = 0 THEN
    bNotAllFramesContainTeachPoints := TRUE;
	END_IF
END_FOR


bNotEnoughTeachPoints := FALSE;
IF    nNumPointsPerSectorT[1] < 2  THEN _ePossibleMode := E_CameraMode.NoCorrection; bNotEnoughTeachPoints := TRUE; //< 2 points in first frame
ELSIF nNumPointsPerSectorT[1] <= 2 THEN _ePossibleMode := E_CameraMode.XYR;          bNotEnoughTeachPoints := TRUE; //< 3 points in first frame
ELSE
  _ePossibleMode := E_CameraMode.Live;
END_IF


// teach is valid
_bTeachOk       := TRUE;
END_METHOD

END_FUNCTION_BLOCK

// ---- POUs/Print/Camera/F_CamPoint_ToString.TcPOU
FUNCTION F_CamPoint_ToString : T_MaxString
VAR_INPUT
  sPoint : ST_CameraPoint;
END_VAR

F_CamPoint_ToString := F_Concat3(
  F_Concat4('id: ', TO_STRING(sPoint.id), ' v: ', SEL(sPoint.valid>0, '0', '1')),
  F_Concat4(' x_ref: ' , TO_STRING(sPoint.x_ref),' y_ref: ', TO_STRING(sPoint.y_ref)),
  F_Concat4(' dx: ' , TO_STRING(sPoint.x),' dy: ', TO_STRING(sPoint.y))
);

END_FUNCTION

// ---- POUs/Print/Camera/F_DeformationPointAcc_ToString.TcPOU
FUNCTION F_DeformationPointAcc_ToString : T_MaxString
VAR_INPUT
  sPointAcc : ST_DeformationPointAccurate;
END_VAR

F_DeformationPointAcc_ToString := F_Concat4(
  F_Concat4('idx: ', TO_STRING(sPointAcc.index), ' v: ', SEL(sPointAcc.valid>0, '0', '1')),
  F_Concat5(' c/r(', TO_STRING(sPointAcc.col), '/', TO_STRING(sPointAcc.row),')'),
  F_Concat4(' x_ref: ' , LREAL_TO_FMTSTR(sPointAcc.x_ref, 4, TRUE),' y_ref: ', LREAL_TO_FMTSTR(sPointAcc.y_ref, 4, TRUE)),
  F_Concat4(' dx: ' , LREAL_TO_FMTSTR(sPointAcc.dx, 4, TRUE),' dy: ', LREAL_TO_FMTSTR(sPointAcc.dy, 4, TRUE))
);

END_FUNCTION

// ---- POUs/Print/Camera/FB_LineCamera106.TcPOU
(*
  QualiVision line camera system
  DMAX106.   
*)
FUNCTION_BLOCK FB_LineCamera106 EXTENDS FB_LineCamera

VAR CONSTANT
  cCameraWidth106           : DINT := 13440;   (*Camera width [px]*)
  cCameraMechOffsetTC106    : REAL :=  88.0;   (*Camera mechanical offset at calibration temp [mm]*)
  cMechOffsetCameraToPU106  : REAL :=  30.31;  (*Camera mechanical offset to PrintUnit [mm]*)
  cPrintUnitMechOffsetTC106 : REAL := 31.4747; (*PrintUnit mechanical offset at calibration temp [mm]*)
END_VAR

SUPER^();

METHOD InitLineCamera
VAR_INPUT
  nPrintUnitResolution         : UDINT;    (*printhead pixel resolution [dpi]*)
  nPrintUnitSubPx              : UDINT;    (*print unit subPixel resolution [SubPx]*)
  nPrintUnitWidth              : UDINT;    (*print unit width in [px]*)
  iCameraTrigger               : I_CameraTrigger;
END_VAR
(*Init for dmax type*)
_nCameraWidth           := cCameraWidth106;
_fCameraMechOffsetTC    := cCameraMechOffsetTC106;
_fMechOffsetCameraToPU  := cMechOffsetCameraToPU106;
_fPrintUnitMechOffsetTC := cPrintUnitMechOffsetTC106;

SUPER^.InitLineCamera( nPrintUnitResolution := nPrintUnitResolution
                      , nPrintUnitSubPx := nPrintUnitSubPx
                      , nPrintUnitWidth := nPrintUnitWidth
                      , iCameraTrigger := iCameraTrigger);
END_METHOD

{attribute 'monitoring':='variable'}
PROPERTY sName : STRING
GET
sName := 'LineCam 106';
END_GET
END_PROPERTY

END_FUNCTION_BLOCK

// ---- POUs/Print/Camera/FB_LineCamera76.TcPOU
(*
  QualiVision line camera system
  DMAX76.   
*)
FUNCTION_BLOCK FB_LineCamera76 EXTENDS FB_LineCamera

VAR CONSTANT
  cCameraWidth76            : DINT :=  9216;   (*Camera width [px]*)
  cCameraMechOffsetTC76     : REAL := 101.5;   (*Camera mechanical offset at calibration temp [mm]*)
  cMechOffsetCameraToPU76   : REAL :=  13.039; (*Camera mechanical offset to PrintUnit [mm]*)
  cPrintUnitMechOffsetTC76  : REAL := 32.9869; (*PrintUnit mechanical offset at calibration temp [mm]*)
END_VAR

SUPER^();

METHOD InitLineCamera
VAR_INPUT
  nPrintUnitResolution         : UDINT;    (*printhead pixel resolution [dpi]*)
  nPrintUnitSubPx              : UDINT;    (*print unit subPixel resolution [SubPx]*)
  nPrintUnitWidth              : UDINT;    (*print unit width in [px]*)
  iCameraTrigger               : I_CameraTrigger;
END_VAR
(*Init for dmax type*)
_nCameraWidth           := cCameraWidth76;
_fCameraMechOffsetTC    := cCameraMechOffsetTC76;
_fMechOffsetCameraToPU  := cMechOffsetCameraToPU76;
_fPrintUnitMechOffsetTC := cPrintUnitMechOffsetTC76;

SUPER^.InitLineCamera( nPrintUnitResolution := nPrintUnitResolution
                      , nPrintUnitSubPx := nPrintUnitSubPx
                      , nPrintUnitWidth := nPrintUnitWidth
                      , iCameraTrigger := iCameraTrigger);
END_METHOD

{attribute 'monitoring':='variable'}
PROPERTY sName : STRING
GET
sName := 'LineCam 76';
END_GET
END_PROPERTY

END_FUNCTION_BLOCK

// ---- POUs/Print/Camera/FB_MarkCamera.TcPOU
(*
  Mark camera system
  2 mark sensors detect sheet marks.   
*)
FUNCTION_BLOCK FB_MarkCamera EXTENDS FB_CameraBase 

VAR_INPUT
  IbSensorState       AT%I* : ARRAY [1..cNbSensors] OF BOOL;        (*Mark sensor state*)
  ItTimeStampPos      AT%I* : ARRAY [1..cNbSensors] OF T_DCTIME64;  (*TimeStamp Pos_Edge @EL1252*)
  ItTimeStampNeg      AT%I* : ARRAY [1..cNbSensors] OF T_DCTIME64;  (*TimeStamp Neg_Edge @EL1252*)

  IfConveyorSpeed           : LREAL;      (*Actual speed of conveyor [m/s]*)
  IfMasterPosition          : LREAL;      (*Master position [µm]*)
END_VAR

VAR
  nCounter                  : UDINT;

  _fSensorDistance          : REAL := 1.0;    (*Distance between the two sensors [m]*)
  _fMarkPositionX           : REAL := 0.010;  (*Distance sheet edge to mark position [m]*)
  _fMarkSizeX               : REAL;           (*Mark size X [mm]*)
  _fMarkSizeY               : REAL;           (*Mark size Y [mm]*)

  tSensorRisingEdge         : ARRAY [1..cNbSensors] OF T_DCTIME64;
  tSensorFallingEdge        : ARRAY [1..cNbSensors] OF T_DCTIME64;
  bMemSensorState           : ARRAY [1..cNbSensors] OF BOOL;       (*Mem mark sensor state*)
  bInhibSensor              : ARRAY [1..cNbSensors] OF BOOL;       (*Inhibit sensor signals, TRUE=inhibit*)
  bSensorStateOK            : ARRAY [1..cNbSensors] OF BOOL;       (*Mark sensor state ok*)
  fSensorDuration           : ARRAY [1..cNbSensors] OF REAL;       (*Sensor signal duration [ns]*)
  fSensorLength             : ARRAY [1..cNbSensors] OF REAL;       (*Sensor signal length [mm]*)
  fS1S2EdgeDistance         : REAL;       (*Edge distance between sensors [mm]*)
  fLateralOffset            : REAL;       (*Lateral offset [mm]*)
  fMemMasterPosition        : LREAL;      (*Mem master position [µm]*)
  bStopCondition            : BOOL;       (*Condition for stop trigger*)
END_VAR

VAR CONSTANT                
  cNbSensors                : UDINT := 2; (*Number of mark sensors*)
END_VAR

IF NOT _bInitialized THEN RETURN; END_IF

(*check parameter*)
IF _fSensorDistance = 0 THEN
	_fSensorDistance := 1.0;
END_IF;

FOR nCounter := 1 TO cNbSensors DO
  (* -------- Detection of rising edge on sensor --------*)
  IF IbSensorState[nCounter] AND NOT bMemSensorState[nCounter] AND NOT bInhibSensor[nCounter] THEN
    tSensorRisingEdge[nCounter] := ItTimeStampPos[nCounter];
    fMemMasterPosition          := IfMasterPosition;
  END_IF;
  
  (* -------- Detection of falling edge --------*)
  IF NOT IbSensorState[nCounter] AND bMemSensorState[nCounter] AND NOT bInhibSensor[nCounter] THEN
    tSensorFallingEdge[nCounter] := ItTimeStampNeg[nCounter];
    fSensorDuration   [nCounter] := LREAL_TO_REAL(ULINT_TO_LREAL(tSensorFallingEdge[nCounter]) - ULINT_TO_LREAL(tSensorRisingEdge[nCounter]));		(* Calculate how long the signal was ON *)
    fSensorLength     [nCounter] := LREAL_TO_REAL(fSensorDuration[nCounter] * IfConveyorSpeed / 1_000_000_000);			(* Calculate the equivalence in mm *)
    bSensorStateOK    [nCounter] := TRUE;   (* now the function can continue to Angle & Offset calculation *)
    bInhibSensor      [nCounter] := TRUE;
  END_IF;
  
  bMemSensorState[nCounter] := IbSensorState[nCounter];			(* Memorization of the sensor1 state for next cycle *)
END_FOR

(* ------------ ANGLE & OFFSET CALCULATION ----------------- *)
IF bSensorStateOK[1] AND bSensorStateOK[2] THEN
  fS1S2EdgeDistance := LREAL_TO_REAL(ULINT_TO_LREAL(tSensorRisingEdge[1] - tSensorRisingEdge[2]) / 1_000_000 * IfConveyorSpeed);	(* Calculate the difference in mm between S1 and S2 trigger *)

  fLateralOffset := (_fMarkSizeY / _fMarkSizeX) * (fSensorLength[1] - fSensorLength[2]) / 2;  (* Evaluation of the offset for each mark *)

  IF _iCameraSink <> 0 THEN
    (*Mark1*)
    stCamPoint.x_ref := F_MeterToSubPixelReal( _fMarkPositionX                                      (*[m]*)
                                              , UDINT_TO_LREAL(_nPrintUnitResolution));             (*Result should be in pixels*)
    stCamPoint.y_ref := F_MeterToSubPixelReal( (_fSubstrateWidth / 2) - (_fSensorDistance / 2)       (*[m]*)
                                              , UDINT_TO_LREAL(_nPrintUnitResolution));             (*Result should be in pixels*)
    stCamPoint.dx    := 0;
    stCamPoint.dy    := F_MeterToSubPixelReal( fLateralOffset * 0.001                              (*[mm] => [m]*)
                                              , UDINT_TO_LREAL(_nPrintUnitResolution));             (*Result should be in pixels*)
    stCamPoint.valid := TRUE;
    
    _iCameraSink.AddCamPoint(stCamPoint);
    _nRxCamPoints := _nRxCamPoints + 1 ;
  
    (*Mark2*)
    stCamPoint.x_ref := F_MeterToSubPixelReal( _fMarkPositionX                                      (*[m]*)
                                             , UDINT_TO_LREAL(_nPrintUnitResolution));             (*Result should be in pixels*)
    stCamPoint.y_ref := F_MeterToSubPixelReal( (_fSubstrateWidth / 2) - (_fSensorDistance / 2) + _fSensorDistance  (*[m]*)
                                             , UDINT_TO_LREAL(_nPrintUnitResolution));             (*Result should be in pixels*)
    stCamPoint.dx    := F_MeterToSubPixelReal( fS1S2EdgeDistance * 0.001                           (*[mm] => [m]*)
                                             , UDINT_TO_LREAL(_nPrintUnitResolution));             (*Result should be in pixels*)
    stCamPoint.dy    := F_MeterToSubPixelReal( fLateralOffset * 0.001                              (*[mm] => [m]*)
                                             , UDINT_TO_LREAL(_nPrintUnitResolution));             (*Result should be in pixels*)
    stCamPoint.valid := TRUE;
    
    _iCameraSink.AddCamPoint(stCamPoint);
    _nRxCamPoints := _nRxCamPoints + 1;
  END_IF;

	bSensorStateOK[1]  := FALSE;
	bSensorStateOK[2]  := FALSE;
END_IF;


(*------------ start and stop signal treatment ------------*)
(*generate stop trigger*)
bStopCondition := (IfMasterPosition >= (fMemMasterPosition + (_fSubstrateLength * 1_000_000)));

IF bStopCondition AND (bInhibSensor[1] OR bInhibSensor[2]) THEN
  bInhibSensor[1] := FALSE;
  bInhibSensor[2] := FALSE;
END_IF;

// TODO: 'implement PUC messages eCPr_PrintMarkError1&2'

{attribute 'monitoring':='call'}
PROPERTY eCameraMode : E_CameraMode
GET
eCameraMode := _eCameraMode;
IF _eCameraMode = E_CameraMode.Auto THEN
  eCameraMode := E_CameraMode.XYR;
END_IF
END_GET
END_PROPERTY

PROPERTY eDeviceType : E_CameraDevice
GET
eDeviceType := E_CameraDevice.PrintMark;
END_GET
END_PROPERTY

PROPERTY fMarkPositionX : REAL
SET
_fMarkPositionX := fMarkPositionX;
END_SET
END_PROPERTY

PROPERTY fMarkSizeX : REAL
SET
_fMarkSizeX := fMarkSizeX;
END_SET
END_PROPERTY

PROPERTY fMarkSizeY : REAL
SET
_fMarkSizeY := fMarkSizeY;
END_SET
END_PROPERTY

PROPERTY fSensorDistance : REAL
SET
_fSensorDistance := fSensorDistance;
END_SET
END_PROPERTY

METHOD GetCamStatus : BOOL
VAR_OUTPUT
  bConnectionOK  : BOOL;    // Camera connected
  bTeachOk       : BOOL;    // Teach successful
  nTeachedPoints : UDINT;   // Teached points for this job
  nScannedPoints : UDINT;   // Scanned points on current sheet
  bCamStarted    : BOOL;    // Camera trigger is active, cam started
  bCamDone       : BOOL;    // Camera finished on last CT
  bErrors        : ARRAY[1..GVL_Camera.nC_NbCamErrors] OF BOOL;  // generic error flag list
END_VAR
bConnectionOK  := TRUE;
bTeachOk       := TRUE; // NO teach availabe
nTeachedPoints := 2;    // 2 marks only
nScannedPoints := _nRxCamPoints;
bCamStarted    := _bCamTriggerStarted;
bCamDone       := _bCamTriggerDone;

GetCamStatus := bConnectionOK AND bTeachOk;   // camera ready
END_METHOD

METHOD InitMarkCamera
VAR_INPUT
  nPrintUnitResolution         : UDINT;    (*printhead pixel resolution [dpi]*)
  nPrintUnitSubPx              : UDINT;    (*print unit subPixel resolution [SubPx]*)
  iCameraTrigger               : I_CameraTrigger;
END_VAR
SUPER^.Init( nPrintUnitResolution      := nPrintUnitResolution
           , nPrintUnitSubPx           := nPrintUnitSubPx
           , iCameraTrigger            := iCameraTrigger
           , bUseCameraTrigger         := FALSE
           , bUseCameraTriggerFeedback := FALSE);

_bInitialized := TRUE;
END_METHOD

(*
  Set mode to camera.
  :return: TRUE if success
*)
METHOD setCameraMode : BOOL
VAR_INPUT
  eCameraMode : E_CameraMode;
END_VAR
IF eCameraMode = E_CameraMode.NoCorrection OR  // supported modi
   eCameraMode = E_CameraMode.XYR THEN
   
  _eCameraMode := eCameraMode;  // set desired mode
  setCameraMode := TRUE;
ELSE
  LogError(F_Concat3('Camera mode=', TO_STRING(eCameraMode), ' not supported by camera'));
  _eCameraMode := E_CameraMode.NoCorrection;
END_IF
END_METHOD

{attribute 'monitoring':='variable'}
PROPERTY sName : STRING
GET
sName := 'Printmarks';
END_GET
END_PROPERTY

END_FUNCTION_BLOCK

// ---- POUs/Print/Camera/FB_SystronCamera.TcPOU
(*
  Systron camera system
  Provides callback function (rx_callback) for received TcpIp messages.   
*)
FUNCTION_BLOCK FB_SystronCamera EXTENDS FB_CameraTcpIp

VAR
  stCameraResult            : ARRAY [1..cNbCameras] OF ST_CAMERA_RESULT;

  nNbTrigger                : INT;
END_VAR

VAR CONSTANT                
  cNbCameras                : UDINT := 2;                (*Number of Systron cameras*)

  cErrorString              : T_MaxString := '<Error(';
  cStartString              : T_MaxString := '<position(';
  cEndingString             : T_MaxString := ');';

  cCameraMinXY              : REAL := -20.0;  (*[mm]*)
  cCameraMaxXY              : REAL := +20.0;  (*[mm]*)
END_VAR

(*Simulation*)
IF _bSimulate THEN
  CreateSimCamPoints();
END_IF

(*
  Simulate camera data
*)
METHOD CreateSimCamPoints : BOOL
VAR_INST
  fbTonTimer    : TON;    (*Send timer*)
  nCounter      : UDINT;  (*Loop counter*)
END_VAR
(*Test points*)
stCameraResult[1].x_ref :=   54;  (*[mm]*)
stCameraResult[1].y_ref := 1003;  (*[mm]*)
stCameraResult[1].valid := TRUE;
stCameraResult[2].x_ref :=   46;  (*[mm]*)
stCameraResult[2].y_ref :=  376;  (*[mm]*)
stCameraResult[2].valid := TRUE;

(*Points are send every 15s*)
fbTonTimer(IN := NOT fbTonTimer.Q, PT := T#15S);
IF fbTonTimer.Q THEN
  FOR nCounter := 1 TO 2 DO
    stCamPoint.x_ref := F_MeterToSubPixelReal( stCameraResult[nCounter].x_ref * 0.001      (*[mm] => [m]*)
                                             , UDINT_TO_LREAL(_nPrintUnitResolution));     (*Result should be in pixels*)
    stCamPoint.y_ref := F_MeterToSubPixelReal( stCameraResult[nCounter].y_ref * 0.001      (*[m]*)
                                             , UDINT_TO_LREAL(_nPrintUnitResolution));     (*Result should be in pixels*)
    stCamPoint.dx    := F_MeterToSubPixelReal( 0.100 * UDINT_TO_REAL(nCounter) * 0.001     (*[mm] => [m]*)
                                            , UDINT_TO_LREAL(_nPrintUnitResolution));     (*Result should be in pixels*)
    stCamPoint.dy    := F_MeterToSubPixelReal( 0.200 * UDINT_TO_REAL(nCounter) * 0.001     (*[mm] => [m]*)
                                            , UDINT_TO_LREAL(_nPrintUnitResolution));     (*Result should be in pixels*)
  
    _iCameraSink.AddCamPoint(stCamPoint);
  END_FOR  
END_IF
END_METHOD

{attribute 'monitoring':='call'}
PROPERTY eCameraMode : E_CameraMode
GET
eCameraMode := _eCameraMode;
IF _eCameraMode = E_CameraMode.Auto THEN
  eCameraMode := E_CameraMode.XYR;
END_IF
END_GET
END_PROPERTY

PROPERTY eDeviceType : E_CameraDevice
GET
eDeviceType := E_CameraDevice.PrintMark;
END_GET
END_PROPERTY

METHOD GetCamStatus : BOOL
VAR_OUTPUT
  bConnectionOK  : BOOL;    // Camera connected
  bTeachOk       : BOOL;    // Teach successful
  nTeachedPoints : UDINT;   // Teached points for this job
  nScannedPoints : UDINT;   // Scanned points on current sheet
  bCamStarted    : BOOL;    // Camera trigger is active, cam started
  bCamDone       : BOOL;    // Camera finished on last CT
  bErrors        : ARRAY[1..GVL_Camera.nC_NbCamErrors] OF BOOL;  // generic error flag list
END_VAR
bConnectionOK  := NOT bConnectionErr OR bSimulate;
bTeachOk       := TRUE; //NO teach availabe (teached by a specific sheet from machine)
nTeachedPoints := 0;
nScannedPoints := 0;
bCamStarted    := _bCamTriggerStarted;
bCamDone       := _bCamTriggerDone;

GetCamStatus := bConnectionOK;
END_METHOD

METHOD rx_callback
VAR_INPUT
	sMessage	: CalmarCompTcpIp.ST_TcpMsg;
END_VAR

VAR
  sAnalyzeLastMessage    : T_MaxString;          (*telegram string*)

  nCounter               : UDINT;
  nFindIndex             : INT;
END_VAR
SUPER^.rx_callback(sMessage := sMessage);

sAnalyzeLastMessage := sLastMessage;

nFindIndex := FIND(sAnalyzeLastMessage, cErrorString);
IF nFindIndex > 0 THEN
  (*Error received*)
  sLastErrorMessage := (DELETE(sAnalyzeLastMessage, (nFindIndex + LEN(cErrorString) - 1), 1));

  (*Extract error message*)
  nFindIndex := FIND(sLastErrorMessage, cEndingString);
  IF nFindIndex > 0 THEN
    sLastErrorMessage := (DELETE(sLastErrorMessage, LEN(sLastErrorMessage) - nFindIndex, nFindIndex));
  END_IF;
ELSE
  (*Search for start string*)
  nFindIndex := FIND(sAnalyzeLastMessage, cStartString);
  IF nFindIndex > 0 THEN
    (*Search string found => remove string to generate index*)
    sAnalyzeLastMessage := (DELETE(sAnalyzeLastMessage, (nFindIndex + LEN(cStartString) - 1), 1));

    (*Search for trigger number*)
    nFindIndex := FIND(sAnalyzeLastMessage, ',');
    IF nFindIndex > 0 THEN
      nNbTrigger := STRING_TO_INT(LEFT(sAnalyzeLastMessage, (nFindIndex - 1)));

      sAnalyzeLastMessage := (DELETE(sAnalyzeLastMessage, nFindIndex, 1));
    END_IF;

    (*Search for rx, ry, v, x and y*)
    FOR nCounter := 1 TO cNbCameras DO
      stCameraResult[nCounter].valid := TRUE;

      (*rx*)
      nFindIndex := FIND(sAnalyzeLastMessage, ',');
      IF nFindIndex > 0 THEN
        stCameraResult[nCounter].x_ref := STRING_TO_REAL(LEFT(sAnalyzeLastMessage, (nFindIndex - 1)));

        IF    (stCameraResult[nCounter].x_ref < cCameraMinXY)
           OR (stCameraResult[nCounter].x_ref > cCameraMaxXY)
        THEN
          stCameraResult[nCounter].valid := FALSE;
        END_IF;

        sAnalyzeLastMessage := (DELETE(sAnalyzeLastMessage, nFindIndex, 1));
      ELSE
        stCameraResult[nCounter].valid := FALSE;
      END_IF;
      (*ry*)
      nFindIndex := FIND(sAnalyzeLastMessage, ',');
      IF nFindIndex > 0 THEN
        stCameraResult[nCounter].y_ref := STRING_TO_REAL(LEFT(sAnalyzeLastMessage, (nFindIndex - 1)));

        IF    (stCameraResult[nCounter].y_ref < cCameraMinXY)
           OR (stCameraResult[nCounter].y_ref > cCameraMaxXY)
        THEN
          stCameraResult[nCounter].valid := FALSE;
        END_IF;

        sAnalyzeLastMessage := (DELETE(sAnalyzeLastMessage, nFindIndex, 1));
      ELSE
        stCameraResult[nCounter].valid := FALSE;
      END_IF;
      (*v*)
      nFindIndex := FIND(sAnalyzeLastMessage, ',');
      IF nFindIndex > 0 THEN
        IF FIND(LEFT(sAnalyzeLastMessage, (nFindIndex - 1)), 'True') > 0 THEN
          stCameraResult[nCounter].valid := TRUE;
        ELSE
          stCameraResult[nCounter].valid := FALSE;
        END_IF;

        sAnalyzeLastMessage := (DELETE(sAnalyzeLastMessage, nFindIndex, 1));
      ELSE
        stCameraResult[nCounter].valid := FALSE;
      END_IF;
      (*x*)
      nFindIndex := FIND(sAnalyzeLastMessage, ',');
      IF nFindIndex > 0 THEN
        stCameraResult[nCounter].x := STRING_TO_REAL(LEFT(sAnalyzeLastMessage, (nFindIndex - 1)));

        IF    (stCameraResult[nCounter].x < cCameraMinXY)
           OR (stCameraResult[nCounter].x > cCameraMaxXY)
        THEN
          stCameraResult[nCounter].valid := FALSE;
        END_IF;

        sAnalyzeLastMessage := (DELETE(sAnalyzeLastMessage, nFindIndex, 1));
      ELSE
        stCameraResult[nCounter].valid := FALSE;
      END_IF;
      (*y*)
      nFindIndex := FIND(sAnalyzeLastMessage, ',');
      IF nFindIndex > 0 THEN
        stCameraResult[nCounter].y := STRING_TO_REAL(LEFT(sAnalyzeLastMessage, (nFindIndex - 1)));

        IF    (stCameraResult[nCounter].y < cCameraMinXY)
           OR (stCameraResult[nCounter].y > cCameraMaxXY)
        THEN
          stCameraResult[nCounter].valid := FALSE;
        END_IF;

        sAnalyzeLastMessage := (DELETE(sAnalyzeLastMessage, nFindIndex, 1));
      ELSE
        nFindIndex := FIND(sAnalyzeLastMessage, ')');
        IF nFindIndex > 0 THEN
          stCameraResult[nCounter].y := STRING_TO_REAL(LEFT(sAnalyzeLastMessage, (nFindIndex - 1)));

          IF    (stCameraResult[nCounter].y < cCameraMinXY)
             OR (stCameraResult[nCounter].y > cCameraMaxXY)
          THEN
            stCameraResult[nCounter].valid := FALSE;
          END_IF;

          sAnalyzeLastMessage := (DELETE(sAnalyzeLastMessage, nFindIndex, 1));
        ELSE
          stCameraResult[nCounter].valid := FALSE;
        END_IF;
      END_IF;
    END_FOR;
  ELSE
    (*Search string not found*)
    FOR nCounter := 1 TO cNbCameras DO
      stCameraResult[nCounter].valid := FALSE;
    END_FOR;
  END_IF;
END_IF;

IF _iCameraSink <> 0 THEN
  FOR nCounter := 1 TO cNbCameras DO
    stCamPoint.x_ref := F_MeterToSubPixelReal( stCameraResult[nCounter].x_ref * 0.001              (*[mm] => [m]*)
                                         , UDINT_TO_LREAL(_nPrintUnitResolution));             (*Result should be in pixels*)
    stCamPoint.y_ref := F_MeterToSubPixelReal( stCameraResult[nCounter].y_ref * 0.001              (*[m]*)
                                         , UDINT_TO_LREAL(_nPrintUnitResolution));             (*Result should be in pixels*)
    stCamPoint.dx    := F_MeterToSubPixelReal( (stCameraResult[nCounter].x_ref - stCameraResult[nCounter].x) * 0.001  (*[mm] => [m]*)
                                         , UDINT_TO_LREAL(_nPrintUnitResolution));             (*Result should be in pixels*)
    stCamPoint.dy    := F_MeterToSubPixelReal( (stCameraResult[nCounter].y_ref - stCameraResult[nCounter].y) * 0.001  (*[mm] => [m]*)
                                         , UDINT_TO_LREAL(_nPrintUnitResolution));             (*Result should be in pixels*)

    _iCameraSink.AddCamPoint(stCamPoint);
  END_FOR
END_IF;

bMsgReceived := FALSE;
END_METHOD

(*
  Set mode to camera.
  :return: TRUE if success
*)
METHOD setCameraMode : BOOL
VAR_INPUT
  eCameraMode : E_CameraMode;
END_VAR
IF eCameraMode = E_CameraMode.NoCorrection OR  // supported modi
   eCameraMode = E_CameraMode.XYR THEN
 
  _eCameraMode := eCameraMode;  // set desired mode
  setCameraMode := TRUE;
ELSE
  LogError(F_Concat3('Camera mode=', TO_STRING(eCameraMode), ' not supported by camera'));
  _eCameraMode := E_CameraMode.NoCorrection;
END_IF
END_METHOD

{attribute 'monitoring':='variable'}
PROPERTY sName : STRING
GET
sName := 'Systron';
END_GET
END_PROPERTY

END_FUNCTION_BLOCK

// ---- POUs/Print/Camera/FB_TcpIpComm.TcPOU
FUNCTION_BLOCK FB_TcpIpComm EXTENDS T_NamedBase IMPLEMENTS I_BootService
VAR_INPUT
END_VAR
VAR_OUTPUT
END_VAR
VAR
  // boot service
  _bStarting       : BOOL := TRUE;
  _tStartDelay     : ARRAY[1..nMaxTcpIpClients] OF TIME;
  fbTonStartDelay  : ARRAY[1..nMaxTcpIpClients] OF TON;
  
  // TcpIp clients list
  sSrvNetId        : T_AmsNetID := '';           (* AmsId of tcpip server.exe, default: empty string. *)
  fbCloseAll       : FB_SocketCloseAll;          (* close all opened sockets *)
  
  fbTcpClients     : ARRAY[1..nMaxTcpIpClients] OF FB_TcpClient;
  pActiveClients   : ARRAY[1..nMaxTcpIpClients] OF POINTER TO FB_TcpClient;
  nActiveTcpClients: UINT;    // active/registered clients¨
  
  nCtr  : UINT;
END_VAR
VAR CONSTANT
  nMaxTcpIpClients      : UINT := 4;
END_VAR

IF _bStarting THEN RETURN; END_IF

// call all active clients
FOR nCtr:=1 TO nActiveTcpClients DO
  fbTonStartDelay[nCtr](IN := TRUE, PT := _tStartDelay[nCtr]);
  IF fbTonStartDelay[nCtr].Q THEN
    fbTcpClients[nCtr](
      //bEnable := .....
      //bConnected => 
    );
  END_IF
END_FOR

PROPERTY bStarting : BOOL
GET
// return booint satus to boot service
bStarting := _bStarting;
END_GET
END_PROPERTY

METHOD closeAllSockets : BOOL
VAR_INST
  bClosing  : BOOL;
END_VAR
(* close all opened/created sockets *)
IF NOT bClosing THEN fbCloseAll( sSrvNetId := sSrvNetId, bExecute:= FALSE ); bClosing := TRUE; END_IF  // be sure to call it once with FALSE

fbCloseAll( sSrvNetId := sSrvNetId, bExecute:= bClosing );
IF NOT fbCloseAll.bBusy THEN
  // done
  //IF fbCloseAll.bError THEN LogError(F_Concat2('CloseAllSockets error=', F_GetAdsErrDescription(lErrCode:=fbCloseAll.nErrId))); 
  //ELSE                      LogInfo('CloseAllSockets done.'); END_IF
  bClosing := FALSE;
END_IF

// return busy
closeAllSockets := fbCloseAll.bBusy;
END_METHOD

METHOD registerTcpIpClient : POINTER TO FB_TcpClient
VAR_INPUT
  sRemoteHost   : ST_SockAddr;
  iHandler      : I_TcpIp_RxMsgHandler;
  tStartDelay   : TIME;
END_VAR

VAR
  pTcpIpClient  : POINTER TO FB_TcpClient;
END_VAR
IF nActiveTcpClients >= nMaxTcpIpClients THEN
  LogError('No free TcpIp client, ignore registerTcpIpClient');
END_IF

nActiveTcpClients := nActiveTcpClients + 1;

// config
fbTcpClients[nActiveTcpClients].sRemoteHost := sRemoteHost.sAddr;
fbTcpClients[nActiveTcpClients].nRemotePort := sRemoteHost.nPort;
_tStartDelay[nActiveTcpClients]             := tStartDelay;

// init
fbTcpClients[nActiveTcpClients].init(
  tReconnect := T#100MS,
  tRxPolling := T#1MS,
  //cMsgTermination := cMSG_TERMINATION_ZERO
);
// start
fbTcpClients[nActiveTcpClients].bEnable := TRUE;
fbTcpClients[nActiveTcpClients].register_RxMsgHandler(bAdd:=TRUE, iHandler);

// return client handle (pointer = full access)
pActiveClients[nActiveTcpClients] := ADR(fbTcpClients[nActiveTcpClients]);
registerTcpIpClient := ADR(fbTcpClients[nActiveTcpClients]);
END_METHOD

METHOD start : BOOL
// called by system boot services, 'regBootService' needed
IF NOT closeAllSockets() THEN
  // done 
  _bStarting := FALSE;  // we are done
END_IF

start := _bStarting;
END_METHOD

END_FUNCTION_BLOCK

// ---- POUs/Print/DefGrid/FB_ContainerDefGrid.TcPOU
FUNCTION_BLOCK FB_ContainerDefGrid EXTENDS FB_ContainerBase
VAR_INPUT
END_VAR
VAR_OUTPUT
END_VAR
VAR
  fBImageDeformation : FB_ImageDeformation;
END_VAR

fBImageDeformation();                       // call run cyclic image deformation

METHOD AbortDeformation : BOOL
VAR_INPUT
  sReason   : STRING;
  Src       : REFERENCE TO T_ErrSrc;
  bHideLog  : BOOL;
END_VAR
IF NOT bHideLog THEN
  LogWarning(F_Concat4('Abort deformation: ', sReason, ' Src: ', Src.aDescr));  // log reason
END_IF
setError(ErrDef:=EC_DefGrid.ecDefGrid_DefGridAbort, Src:=Src); // tag ct as error
fBImageDeformation.abort();  // abort deformation
StopScript(iCT:=THIS^);
END_METHOD

METHOD AddCamPoint : BOOL
VAR_INPUT
  sPoint : ST_DeformationPointAccurate;
END_VAR
AddCamPoint := fBImageDeformation.addCamPoint(sNewPoint:=sPoint);
END_METHOD

PROPERTY bLimited : BOOL
GET
bLimited := fBImageDeformation.bDeformationGridLimited;
END_GET
SET
fBImageDeformation.bDeformationGridLimited := bLimited;
END_SET
END_PROPERTY

(*
  Create a container, build very basics.
*)
METHOD Create : BOOL
VAR_INPUT
	nCTId	            : DINT;     (* a container identifier *)
	nCTIndex	        : UDINT;	  (* memory index (array index if CT in CT array) *)
END_VAR
SUPER^.Create(nCTId:=nCTId, nCTIndex:=nCTIndex);
fBImageDeformation.reset();
fBImageDeformation.nProcessId := THIS^.pCT^.iId;
END_METHOD

PROPERTY eCamMode : E_CameraMode
GET
eCamMode := fBImageDeformation.eCamMode;
END_GET
END_PROPERTY

(*
  Shift in x [SubPx]
*)
PROPERTY fDxShift : LREAL
GET
VAR
  errCtr : UDINT;
END_VAR
fDxShift := fBImageDeformation._nDxShift;
END_GET
END_PROPERTY

(*
  Shift in y [Px]
*)
PROPERTY fDyShift : LREAL
GET
VAR
  errCtr : UDINT;
END_VAR
fDyShift := fBImageDeformation._nDyShift;
END_GET
END_PROPERTY

PROPERTY fPrintLengthEffective : LREAL
GET
fPrintLengthEffective := fBImageDeformation.fPrintLengthEffective;
END_GET
SET
fBImageDeformation.fPrintLengthEffective := fPrintLengthEffective;
END_SET
END_PROPERTY

(*
  get a deformation point.
  :returns: TRUE if successful
*)
METHOD getDeformationPoint : BOOL;
VAR_INPUT
  nCol : UDINT;   // col select
  nRow : UDINT;   // row select
  nSel : UDINT;   // table selection
END_VAR
VAR_OUTPUT
  sPoint : ST_DeformationPointAccurate;
  bWasSet : BOOL;           // point was set by deformation
END_VAR
getDeformationPoint := fBImageDeformation.getDeformationPoint(nCol:=nCol, nRow:=nRow, nSel:=nSel, sPoint=>sPoint, bWasSet=>bWasSet);
END_METHOD

(*
  Deformation state of CT.
  :return:  TRUE in case of error -> any deformation error
*)
METHOD getDeformationStatus : BOOL
VAR_INPUT
END_VAR
VAR_OUTPUT
  eDStep: E_DeformationStep;// deformation step
  bDone : BOOL;             // deformation done
  bBusy : BOOL;             // deformation is busy
  nErrorId : UDINT;         // error id in case of error
  tExecutionTime : TIME;    // script update execution time?
  bAborted : BOOL;          // deformation is aborted/error
END_VAR
getDeformationStatus := fBImageDeformation.bError;

eDStep:= fBImageDeformation.eStep;
bBusy := fBImageDeformation.bBusy;
bDone := fBImageDeformation.bDone;
nErrorId := fBImageDeformation.nErrorId;
tExecutionTime := fBImageDeformation.tExecutionTime;
bAborted := fBImageDeformation.bAborted;
END_METHOD

PROPERTY LogLevel : E_LogSeverity
GET
LogLevel := SUPER^.LogLevel;
END_GET
SET
fBImageDeformation.LogLevel := LogLevel;
SUPER^.LogLevel := LogLevel;
END_SET
END_PROPERTY

PROPERTY nAvailableGridCols : UDINT
GET
nAvailableGridCols := fBImageDeformation._nGridCols;
END_GET
END_PROPERTY

PROPERTY nAvailableGridPoints : UDINT
GET
nAvailableGridPoints := fBImageDeformation.nAvailableGridPoints;
END_GET
END_PROPERTY

PROPERTY PUBLIC nRegisteredCameraPoints : UDINT
GET
nRegisteredCameraPoints := fBImageDeformation._nCamPoints;
END_GET
END_PROPERTY

PROPERTY pImageDeformation : POINTER TO FB_ImageDeformation
GET
pImageDeformation := ADR(fBImageDeformation);
END_GET
END_PROPERTY

PROPERTY sDefGridSettings : ST_DefGridSettings
GET
sDefGridSettings := fBImageDeformation.sDefGridSettings;
END_GET
END_PROPERTY

METHOD StartCamera
VAR_INPUT
  eCameraMode  : E_CameraMode;   // used camera mode
  fFeatureGrid : LREAL;          // deformation module update interval [Px]
  bResetDeformation : BOOL;      // reset current deformation state
END_VAR
// reset old deformation
IF bResetDeformation THEN
  fBImageDeformation.reset();
END_IF

// update mode
fBImageDeformation.eCamMode := eCameraMode;
fBImageDeformation.fFeatureGrid := fFeatureGrid;
fBImageDeformation.eStep := E_DeformationStep.cameraStarted;
END_METHOD

METHOD StartDeformation
VAR_INPUT
  sDefGridSettings : ST_DefGridSettings;
  fStartDeformationPos : LREAL;   // reference start position in [px]
END_VAR
fBImageDeformation.sDefGridSettings := sDefGridSettings;                  // apply grid setting
fBImageDeformation.startDeformation(                                      // start deformation process
  fStartDefPos:=fStartDeformationPos,     // reference position at current position [Px]
  fImageLength:=pJob^.fImageDepth / 1000        // fSubstrateDepth            //update with intended length
);
END_METHOD

METHOD StartScript
VAR_INPUT
  iDeformationHandler : I_DeformationHandler;
END_VAR
fBImageDeformation.iDeformationHandler := iDeformationHandler;
fBImageDeformation.eStep := E_DeformationStep.createdScriptContainer;
END_METHOD

METHOD StopScript : BOOL
VAR_INPUT
  iCT : I_CT;
END_VAR
IF fBImageDeformation.iDeformationHandler <> 0 THEN
  fBImageDeformation.iDeformationHandler.DeleteCachedCt(iCT:=iCT);
  fBImageDeformation.iDeformationHandler := 0; // remove handler after stopping (prevent further calls on same CT)
END_IF
END_METHOD

(*
  save a streamed deformation point.
  :returns: TRUE if successful
*)
METHOD storeStreamedDeformationPoint : BOOL;
VAR_INPUT
  pPoint : POINTER TO ST_DeformationPointAccurate;
END_VAR
IF pPoint = 0 THEN RETURN; END_IF

storeStreamedDeformationPoint := fBImageDeformation.storeStreamedDeformationPoint(pPoint:=pPoint);
END_METHOD

METHOD UpdateDeformation
VAR_INPUT
  fPos : LREAL; // relative deformation position in [px]
END_VAR
fBImageDeformation.updateDeformation(fPos:=fPos);
END_METHOD

END_FUNCTION_BLOCK

// ---- POUs/Print/DefGrid/FB_ImageDeformation.TcPOU
FUNCTION_BLOCK FB_ImageDeformation EXTENDS FB_PythonDeformation
VAR
  _eDeformationStep : E_DeformationStep;    // current active deformation step (handler)
  _eCameraMode      : E_CameraMode;         // active deformation mode
  _fFeatureGrid     : LREAL;                // camera feature grid [Px]
  _iDefHandler      : I_DeformationHandler; // deformation handler interface for global deformation control
  _nImgProcPoints   : DINT;                 // to calc gloabl dx/dy
  _nDxShift, _nDxSum : LREAL;               // global x grid shift
  _nDyShift, _nDySum : LREAL;               // global y grid shift
  
  // Cam points (stored locally)
  _nCamPoints        : UDINT;
  _sCamPoints        : ARRAY[0..100] OF ST_CameraPointTbl;   // received cam points
  _nCamPoint_MaxRefX : LREAL;               // max. x position of all available cam points [px]

  _sDefGridSettings  : ST_DefGridSettings;  // local copy of settings  
  // local DefGrid table [calculated]
  _sDefGridPoints    : ARRAY[0..nMAX_COLS_DEFGRID, 0..nMAX_ROWS_DEFGRID] OF ST_DeformationPointTbl; // [col, row] local grid point table
  _nGridPoints       : UDINT;               // stored and available grid points
  _nGridCols         : UDINT;               // count current complete grid columns
  // local DefGrid table [streamed]
  _sDefGridPointsStreamed : ARRAY[0..nMAX_COLS_DEFGRID, 0..nMAX_ROWS_DEFGRID] OF ST_DeformationPointTbl; // [col, row] local grid point table 
  _nGridRowsStreamed, _nGridColsStreamed : UDINT;
  
  // local grid handler(s) helper
  _nLocalGridColsGenerated: UDINT;          // already generated "local" grid columns XYR [0..x]

  _fStartDeformPos  : LREAL;                // position [Px] where deformation started on ct
  _nUpdatedGridCol  : UDINT;                // already updated grid column
  _nUpdatedFeature  : UDINT;                // number of updated features (a distance)
  _fPrintLengthOriginal  : LREAL;           // intended image depth in [m]
  _fPrintLengthEffective : LREAL;           // effective detected printing length in [m] (not yet used, but could be used for more accureate dx calculation in the future)
  _bDeformationGridLimited : BOOL;              // some deformation points were limited to a min/max boundary
  // others
  _nErrorId         : UDINT := 0;
  _sTempPoint       : ST_DeformationPointAccurate; 
END_VAR
VAR_STAT
  // sim
  eTestGridSelection : E_GridTypeSelection;
  nTestGridFactor : LREAL := 20;
END_VAR
VAR CONSTANT
  tPYTHON_TIMEOUT   : TIME  := T#500MS;     // python deformation script update response timeout  
  nMAX_COLS_DEFGRID : UDINT := 100;         // if you update this value you need to update the array variables as well (there we can't use this constant (beckhoff bug in table view))
  nMAX_ROWS_DEFGRID : UDINT := 100;         // if you update this value you need to update the array variables as well (there we can't use this constant (beckhoff bug in table view))
  nMAX_CAM_POINTS   : UDINT := 100;         // if you update this value you need to update the array variables as well (there we can't use this constant (beckhoff bug in table view))
END_VAR

IF NOT bInitialized THEN
  init();
END_IF

IF bUsePy THEN
  ExecPy();       // call python deformation handler
  
  // pull all GridPoints from FIFO and store to local table
  WHILE PopDeformationPoint(sNewPoint=>_sTempPoint) DO
    storeDeformationPoint(sPoint:=_sTempPoint);    // save point to table
  END_WHILE
END_IF

METHOD abort : BOOL
VAR_INPUT
END_VAR
_bAborted := TRUE;
END_METHOD

METHOD addCamPoint : BOOL
VAR_INPUT
  sNewPoint : ST_DeformationPointAccurate;
END_VAR
VAR
  sPointPx  : ST_DeformationPoint;
END_VAR
IF bUsePy THEN
  // push point to fifo for script
  
  addCamPoint := PushDeformationPoint(
                      sPoint:=F_EncodeDeformationPoint(sPoint:=sNewPoint, nResolution:=GVL_Deformation.nC_GridSubReso)
                 );
ELSE
  addCamPoint := TRUE;
END_IF

// store it to local table
IF addCamPoint THEN
  storeCameraPoint(sPoint:=sNewPoint); // store locally
END_IF
END_METHOD

PROPERTY bAborted : BOOL
GET
bAborted := _bAborted;
END_GET
END_PROPERTY

PROPERTY bBusy : BOOL
GET
bBusy := bPythonBusy AND NOT _bAborted;
END_GET
END_PROPERTY

PROPERTY bDeformationGridLimited : BOOL
GET
bDeformationGridLimited := _bDeformationGridLimited;
END_GET
SET
_bDeformationGridLimited := bDeformationGridLimited;
END_SET
END_PROPERTY

PROPERTY bDone : BOOL
GET
bDone := bPythonDeformationDone OR _bAborted OR (eStep = E_DeformationStep.nothing);
END_GET
END_PROPERTY

PROPERTY bError : BOOL
GET
bError := bPythonError OR _bAborted;
END_GET
END_PROPERTY

PROPERTY PRIVATE bUsePy : BOOL
GET
IF _sDefGridSettings.eDeformationType=E_DeformationType.ScriptGrid OR _sDefGridSettings.eDeformationType = E_DeformationType.ScriptGridTrend THEN
  bUsePy := TRUE;
END_IF
END_GET
END_PROPERTY

METHOD dumpGrid : BOOL
VAR_INPUT
END_VAR
END_METHOD

PROPERTY eCamMode : E_CameraMode
GET
eCamMode := _eCameraMode;
END_GET
SET
_eCameraMode := eCamMode;
END_SET
END_PROPERTY

PROPERTY eStep : E_DeformationStep
GET
eStep := _eDeformationStep;
END_GET
SET
IF eStep > _eDeformationStep THEN
  LogLvl(Lvl:=E_LogSeverity.Detail, Msg:=F_Concat4('Change deformation step: ', TO_STRING(_eDeformationStep), '->', TO_STRING(eStep)));
  _eDeformationStep := eStep;
END_IF
END_SET
END_PROPERTY

(*
  Camera feature grid. Section distance where points are detected and sent as group to PLC.
*)
PROPERTY fFeatureGrid : LREAL
GET
fFeatureGrid := _fFeatureGrid;
END_GET
SET
_fFeatureGrid := fFeatureGrid;
END_SET
END_PROPERTY

PROPERTY fPrintLengthEffective : LREAL
GET
fPrintLengthEffective := _fPrintLengthEffective;
END_GET
SET
_fPrintLengthEffective := fPrintLengthEffective;
END_SET
END_PROPERTY

// get neighbour camera point
// :returns: TRUE if present
METHOD PRIVATE getCamNeighbourPoint : BOOL
VAR_INPUT
  fPos    : LREAL;   // [px]
  nOffset : DINT;    // 0=previous, 1=next
END_VAR
VAR_OUTPUT
  Pn : ST_CameraPointTbl;
END_VAR
VAR
  i : DINT;
  foundIdx : DINT;
END_VAR
foundIdx := -1;
FOR i:=0 TO TO_DINT(_nCamPoints)-1 DO
  // previous search
  IF nOffset = 0 THEN
    IF _sCamPoints[i].sPoint.x_ref <= fpos THEN
      foundIdx := i;
    ELSE
      EXIT;
    END_IF
    
  // next searchs  
  ELSIF nOffset = 1 THEN
    IF _sCamPoints[i].sPoint.x_ref > fpos THEN
      foundIdx := i;
      EXIT;
    END_IF
  END_IF
END_FOR

IF foundIdx >= 0 THEN
  Pn := _sCamPoints[foundIdx];
  getCamNeighbourPoint := TRUE;  
END_IF
END_METHOD

// get neighbour camera point
// :returns: TRUE if present
METHOD getCamPointX : BOOL
VAR_INPUT
  nIdx : UDINT;    // 0=last, 1=first, 2=second
END_VAR
VAR_OUTPUT
  Pn : ST_CameraPointTbl;
END_VAR
IF nIdx = 0 THEN
  Pn := _sCamPoints[_nCamPoints-1];  // return first cam point
  getCamPointX := TRUE;
ELSIF nIdx <= _nCamPoints THEN
  Pn := _sCamPoints[nIdx-1];
  getCamPointX := TRUE;
ELSE
  //error
  Pn := _sCamPoints[0];   // error return first as fallback 
END_IF
END_METHOD

(*
  get a deformation point.
  :returns: TRUE if successful
*)
METHOD getDeformationPoint :  BOOL;
VAR_INPUT
  nCol : UDINT;   // col select
  nRow : UDINT;   // row select
  nSel : UDINT;   // table selection 0=GeneratedGrid, 1=StreamedGrid
END_VAR
VAR_OUTPUT
  sPoint : ST_DeformationPointAccurate;
  bWasSet : BOOL;
END_VAR
getDeformationPoint := FALSE;

IF TO_UDINT(nCol) > nMAX_COLS_DEFGRID THEN LogError(F_Concat5('getDeformationPoint: point col=', TO_STRING(nCol), ' out of table > ', TO_STRING(nMAX_COLS_DEFGRID), '')); RETURN; END_IF
IF TO_UDINT(nRow) > nMAX_ROWS_DEFGRID THEN LogError(F_Concat5('getDeformationPoint: point row=', TO_STRING(nRow), ' out of table > ', TO_STRING(nMAX_ROWS_DEFGRID), '')); RETURN; END_IF

IF nSel = 1 THEN
  sPoint  := _sDefGridPointsStreamed[nCol, nRow].sPoint;
  bWasSet := _sDefGridPointsStreamed[nCol, nRow].bSet;  
ELSE
  sPoint  := _sDefGridPoints[nCol, nRow].sPoint;
  bWasSet := _sDefGridPoints[nCol, nRow].bSet;  
END_IF

getDeformationPoint := TRUE;
END_METHOD

METHOD PROTECTED gridImgProc
VAR_INPUT
  pNewDeformationPoint	: POINTER TO ST_DeformationPointAccurate;
END_VAR
IF pNewDeformationPoint = 0 THEN RETURN; END_IF

_nDxSum := (_nDxSum + pNewDeformationPoint^.dx);
_nDySum := (_nDySum + pNewDeformationPoint^.dy);
IF _nImgProcPoints > 0 THEN
  _nDxShift := _nDxSum / _nImgProcPoints;
  _nDyShift := _nDySum / _nImgProcPoints;
END_IF
_nImgProcPoints := _nImgProcPoints + 1;
END_METHOD

PROPERTY iDeformationHandler : I_DeformationHandler
GET
iDeformationHandler := _iDefHandler;
END_GET
SET
_iDefHandler := iDeformationHandler;
END_SET
END_PROPERTY

METHOD init
VAR_INPUT
END_VAR
_fbTimeout.PT := tPYTHON_TIMEOUT;
bInitialized := TRUE;
END_METHOD

PROPERTY nAvailableCamPoints : UDINT
GET
nAvailableCamPoints := _nCamPoints;
END_GET
END_PROPERTY

PROPERTY nAvailableGridPoints : UDINT
GET
nAvailableGridPoints := _nGridPoints;
END_GET
END_PROPERTY

PROPERTY nErrorId : UDINT
GET
nErrorId := _nErrorId;
END_GET
END_PROPERTY

PROPERTY nProcessId : DINT
GET
nProcessId := nPythonId;
END_GET
SET
nPythonId := nProcessId;
END_SET
END_PROPERTY

METHOD reset
VAR_INPUT
END_VAR
SUPER^.Reset();   // reset FB_PythonDeformation

_nGridPoints := 0;
_nGridCols := 0;
_nCamPoints := 0;
_nCamPoint_MaxRefX := 0;
MEMSET(destAddr:=ADR(_sDefGridPoints), fillByte:=0, n:=SIZEOF(_sDefGridPoints));
MEMSET(destAddr:=ADR(_sCamPoints), fillByte:=0, n:=SIZEOF(_sCamPoints));
MEMSET(destAddr:=ADR(_sDefGridSettings), fillByte:=0, n:=SIZEOF(_sDefGridSettings));

MEMSET(destAddr:=ADR(_sDefGridPointsStreamed), fillByte:=0, n:=SIZEOF(_sDefGridPointsStreamed));
_nGridRowsStreamed := 0;
_nGridColsStreamed := 0;

_eDeformationStep := E_DeformationStep.nothing;
_eCameraMode := E_CameraMode.NoCorrection;
_iDefHandler := 0;
_nImgProcPoints   := 0;
_nDxShift         := 0;
_nDyShift         := 0;
_nDxSum           := 0;
_nDySum           := 0; 

_nLocalGridColsGenerated:=0;
_fStartDeformPos:=0;
_nUpdatedGridCol := 0;
_nUpdatedFeature := 0;
_nErrorId := 0;
_tExecutionTime := T#0s;
END_METHOD

PROPERTY sDefGridSettings : ST_DefGridSettings
GET
sDefGridSettings := _sDefGridSettings;
END_GET
SET
_sDefGridSettings := sDefGridSettings;
END_SET
END_PROPERTY

METHOD startDeformation
VAR_INPUT
  fStartDefPos : LREAL;  // [Px]
  fImageLength : LREAL;  // [m] original image length
END_VAR
_fStartDeformPos := fStartDefPos;
_fPrintLengthOriginal := fImageLength;
_fPrintLengthEffective := fImageLength;
_nUpdatedGridCol := 0;
_nUpdatedFeature := 0;
_nCamPoint_MaxRefX := 0;

eStep := E_DeformationStep.gridStarted;  // signal to start deformation (update process)
END_METHOD

METHOD PRIVATE storeCameraPoint
VAR_INPUT
  sPoint : ST_DeformationPointAccurate;
END_VAR
// save point with checks and log.

//-- check table overflow
IF _nCamPoints >= nMAX_CAM_POINTS THEN LogError(F_Concat3('storeCamPoint: array overflow ', TO_STRING(_nCamPoints), ' ignore point, ')); RETURN; END_IF

//-- store point
_sCamPoints[_nCamPoints].bSet := TRUE;
_sCamPoints[_nCamPoints].sPoint := sPoint;
_sCamPoints[_nCamPoints].tTime := F_GetCurDcTaskTime64();
_nCamPoints := _nCamPoints+1;

// -- max. x pos 
IF sPoint.x_ref > _nCamPoint_MaxRefX THEN
  _nCamPoint_MaxRefX := sPoint.x_ref;  // point most far in ct
END_IF
END_METHOD

METHOD PRIVATE storeDeformationPoint
VAR_INPUT
  sPoint : ST_DeformationPointAccurate;
END_VAR
// do global point img processing
gridImgProc(pNewDeformationPoint:=ADR(sPoint));

// save point with checks and log.
//-- check table overflow
IF TO_UDINT(sPoint.col) > nMAX_COLS_DEFGRID THEN LogError(F_Concat5('point col=', TO_STRING(sPoint.col), ' exceeds max=', TO_STRING(nMAX_COLS_DEFGRID), ' ignore point')); RETURN; END_IF
IF TO_UDINT(sPoint.row) > nMAX_ROWS_DEFGRID THEN LogError(F_Concat5('point row=', TO_STRING(sPoint.row), ' exceeds max=', TO_STRING(nMAX_ROWS_DEFGRID), ' ignore point')); RETURN; END_IF
  
//-- store point
_sDefGridPoints[sPoint.col, sPoint.row].bSet := TRUE;
_sDefGridPoints[sPoint.col, sPoint.row].sPoint := sPoint;
_sDefGridPoints[sPoint.col, sPoint.row].tTime := F_GetCurDcTaskTime64();
IF sPoint.x_ref = 0 THEN _sDefGridPoints[sPoint.col, sPoint.row].sPoint.x_ref := sPoint.col * TO_DINT(_sDefGridSettings.nGridPitchX); END_IF// calc x pos of grid point (if not done by script)
IF sPoint.y_ref = 0 THEN _sDefGridPoints[sPoint.col, sPoint.row].sPoint.y_ref := sPoint.row * TO_DINT(_sDefGridSettings.nGridPitchY); END_IF// calc x pos of grid point (if not done by script)
// count grid points 
_nGridPoints := _nGridPoints + 1;
// count current complete grid columns
IF _sDefGridSettings.nGridSizeY > 0 THEN
  _nGridCols := (_nGridPoints/_sDefGridSettings.nGridSizeY);
END_IF
END_METHOD

METHOD storeStreamedDeformationPoint : BOOL
VAR_INPUT
  pPoint : POINTER TO ST_DeformationPointAccurate;
END_VAR
IF pPoint = 0 THEN RETURN; END_IF
IF TO_UDINT(pPoint^.col) > nMAX_COLS_DEFGRID THEN RETURN; END_IF
IF TO_UDINT(pPoint^.row) > nMAX_ROWS_DEFGRID THEN RETURN; END_IF

_sDefGridPointsStreamed[pPoint^.col, pPoint^.row].bSet := TRUE;
_sDefGridPointsStreamed[pPoint^.col, pPoint^.row].sPoint := pPoint^;
_sDefGridPointsStreamed[pPoint^.col, pPoint^.row].tTime := F_GetCurDcTaskTime64();
IF pPoint^.x_ref = 0 THEN _sDefGridPointsStreamed[pPoint^.col, pPoint^.row].sPoint.x_ref := pPoint^.col * TO_DINT(_sDefGridSettings.nGridPitchX); END_IF// calc x pos of grid point (if not done by script)
IF pPoint^.y_ref = 0 THEN _sDefGridPointsStreamed[pPoint^.col, pPoint^.row].sPoint.y_ref := pPoint^.row * TO_DINT(_sDefGridSettings.nGridPitchY); END_IF// calc x pos of grid point (if not done by script)
_nGridColsStreamed := MAX(_nGridColsStreamed, TO_UDINT(pPoint^.col));
_nGridRowsStreamed := MAX(_nGridRowsStreamed, TO_UDINT(pPoint^.row));

storeStreamedDeformationPoint := TRUE;
END_METHOD

PROPERTY tExecutionTime : TIME
GET
tExecutionTime := _tExecutionTime;  // TODO: in case of local processor read other execution time
END_GET
END_PROPERTY

METHOD updateDeformation
VAR_INPUT
  fPos : LREAL;  // current CT position in [px]
END_VAR
VAR
  fPosRel_Deform      : LREAL;    // position relative to start deformation [px]
  fPosRel_CamFeature  : LREAL;    // theoretical feature position [feature nr](based on StartDeformation NOT real on camera)
  fPosRel_GridCol     : LREAL;    // current deformation grid number [grid nr]
  sPoint : ST_DeformationPoint;
  nCurrentCol, nCurrentFeature : UDINT;
END_VAR
// cyclic call and update deformation script
// - parameter checks
IF eStep < E_DeformationStep.gridStarted OR bDone THEN RETURN; END_IF  // nothing to do if deformation was not started
IF _sDefGridSettings.nGridSizeX = 0 THEN RETURN; END_IF
IF fFeatureGrid = 0 THEN fFeatureGrid := 1024; END_IF         // set some valid default (prevents division crash)

// - calc relative Deformation position
fPosRel_Deform     := fPos - _fStartDeformPos;
fPosRel_CamFeature := fPosRel_Deform / _fFeatureGrid;
fPosRel_GridCol    := fPosRel_Deform / _sDefGridSettings.nGridPitchX;

// - check available cam points --> current feature
//    Is this blocking when position is retracting?
IF FLOOR(fPosRel_CamFeature) > _nUpdatedFeature   // by CameraFeature pitch (to sync with reception of cam points)
   //FLOOR(fPosRel_GridCol) > _nUpdatedGridCol    // by Grid Pitch  // AND _nUpdatedGridCol <= _sDefGridSettings.nGridSizeX
THEN

  nCurrentCol := TO_UDINT(FLOOR(fPosRel_GridCol));
  nCurrentFeature :=  TO_UDINT(FLOOR(fPosRel_CamFeature));

  // debug info
  LogLvl(Lvl:=E_LogSeverity.Debug, Msg:=
    F_Concat6(
        F_Concat2('update at: ', TO_STRING(fPosRel_Deform)),
        F_Concat3(' feature(', TO_STRING(fPosRel_CamFeature), ')'),
        F_Concat2(' CamP: ', TO_STRING(_nCamPoints)),
        F_Concat2(' maxX: ', TO_STRING(_nCamPoint_MaxRefX)),
        F_Concat2(' GridP: ', TO_STRING(_nGridPoints)),
        F_Concat2(' at Col: ', TO_STRING(nCurrentCol))
    )
  );

  // - update Grid (py or local) with desired position
  IF bUsePy THEN
    IF _nCamPoints > 2 THEN
      UpdatePy(fPosition:=fPosRel_Deform);
      _nUpdatedGridCol := nCurrentCol;
      _nUpdatedFeature := nCurrentFeature;
    END_IF
  ELSIF _sDefGridSettings.eDeformationType = E_DeformationType.LocalMarks1D THEN
    updateLocal_1D_Marks(nGridCol:=nCurrentCol, nFeatureCt:=nCurrentFeature);
    _nUpdatedGridCol := nCurrentCol;
    _nUpdatedFeature := nCurrentFeature;
  END_IF
END_IF
END_METHOD

METHOD PRIVATE updateLocal_1D_Marks : BOOL
VAR_INPUT
  nGridCol : UDINT;
  nFeatureCt : UDINT;
END_VAR
VAR
  row, col : UDINT;
  ct : DINT;
  col_pos_px : LREAL;   // column position in [px]
  sTmpPoint : ST_DeformationPointAccurate;
  dx, dy : LREAL;
  generateGridForCol : BOOL;
  Pn0, Pn1 : ST_CameraPointTbl;
  pPx : POINTER TO ST_CameraPointTbl;
  bn0, bn1 : BOOL;
  bFirstCol, bLastCol : BOOL;
  fPointDist : LREAL;
  relativePosX : LREAL;
END_VAR
VAR_INST
  fTrig_Done : F_TRIG;
END_VAR
VAR CONSTANT
  fC_SignConversion : LREAL := -1; 
END_VAR
bFirstCol := SEL(nGridCol=0, FALSE, TRUE);
bLastCol  := SEL(nGridCol=_sDefGridSettings.nGridSizeX-1, FALSE, TRUE);

ct := 0;
FOR col:=_nLocalGridColsGenerated TO nGridCol DO      // loop over not yet gnerated columns 
  LogLvl(Lvl:=E_LogSeverity.Debug, Msg:= F_Concat2(F_Concat2('check grid for col: ', TO_STRING(col)), ''));
  
  col_pos_px := col * _sDefGridSettings.nGridPitchX;
  dx:=0; dy:=0;
  
  bn0 := getCamNeighbourPoint(fPos:=col_pos_px, nOffset:=0, Pn=>Pn0);
  bn1 := getCamNeighbourPoint(fPos:=col_pos_px, nOffset:=1, Pn=>Pn1);
  
  IF bn0 AND bn1 THEN
    // we have neighbour points --> interpolate displacement inbetween
    // dx/dy interpolation between previous and next cam point
    fPointDist := Pn1.sPoint.x_ref-Pn0.sPoint.x_ref;
    fPointDist := SEL(fPointDist=0, fPointDist, 1);    // avoid 0 division crash
    relativePosX := (col_pos_px-Pn0.sPoint.x_ref) / (fPointDist);    // relative position of col between two cam points
    dx := fC_SignConversion * (Pn0.sPoint.dx + (Pn1.sPoint.dx - Pn0.sPoint.dx) * relativePosX);
    dy := fC_SignConversion * (Pn0.sPoint.dy + (Pn1.sPoint.dy - Pn0.sPoint.dy) * relativePosX);
    generateGridForCol:=TRUE;
    
  ELSIF bFirstCol THEN
    // generate first col when we have a cam point -> deformation from first point
    IF    bn0 THEN dx:=fC_SignConversion*Pn0.sPoint.dx; dy:=fC_SignConversion*Pn0.sPoint.dy; generateGridForCol:=TRUE;
    ELSIF bn1 THEN dx:=fC_SignConversion*Pn1.sPoint.dx; dy:=fC_SignConversion*Pn1.sPoint.dy; generateGridForCol:=TRUE;
    END_IF
    
  ELSE
    // not framed by two points toward the end, purge colums if no valid cam point is given next
    IF nGridCol - _nLocalGridColsGenerated >= 3 OR bLastCol THEN 
      IF _nCamPoints > 1 THEN
        // calc deformation based on first and last point
        bn0 := getCamPointX(nIdx:=1, Pn=>Pn0);  // first
        bn0 := getCamPointX(nIdx:=0, Pn=>Pn1);  // last
        fPointDist := Pn1.sPoint.x_ref-Pn0.sPoint.x_ref;      // distance of the two points
        fPointDist := SEL(fPointDist=0, fPointDist, 1);                // avoid 0 division crash
        relativePosX := (col_pos_px-Pn0.sPoint.x_ref) / (fPointDist);    // relative position of col between two cam points
        dx := fC_SignConversion * (Pn0.sPoint.dx + (Pn1.sPoint.dx - Pn0.sPoint.dx) * relativePosX);
        dy := fC_SignConversion * (Pn0.sPoint.dy + (Pn1.sPoint.dy - Pn0.sPoint.dy) * relativePosX);
      ELSE
        // repeat first correction (we do not have more information)
        pPx := SEL(bn1, ADR(Pn0), ADR(Pn1));
        dx := fC_SignConversion * pPx^.sPoint.dx;
        dy := fC_SignConversion * pPx^.sPoint.dy;
      END_IF
      
      generateGridForCol := TRUE;
    END_IF    
  END_IF
  
  // SIMULATION: some test grid (overwrite calculation)
  IF eTestGridSelection <> E_GridTypeSelection.Default THEN
    CASE eTestGridSelection OF
      0: dx := dx; dy := dy;                                        // default usekeep calculated
      1: dx := dy := 0;                                             // no deformation on ct 
      2: dx := nTestGridFactor; dy := 0;                            // dx static (Factor)
      3: dx := 0; dy := nTestGridFactor;                            // dy static (Factor)
      4: dx := 0; dy := TO_LREAL(col) * nTestGridFactor;            // dx = factor * col
      5: dx := TO_LREAL(col) * nTestGridFactor; dy := 0;            // dy = factor * col
      6: dx := SEL(row=1, 0, nTestGridFactor ); dy := 0;            // dx row 1 = factor ( test BOF)
    END_CASE
    generateGridForCol := TRUE;
  END_IF  
  
  // generate grid for column  
  IF generateGridForCol THEN
    LogLvl(Lvl:=E_LogSeverity.Debug, Msg:= F_Concat6('generate grid for col: ', TO_STRING(col), ' dx=', TO_STRING(dx), '/dy=', TO_STRING(dy)));

    // check for cam points and generate grid
    FOR row:=0 TO _sDefGridSettings.nGridSizeY -1 DO    // all points per col
      //LogLvl(Lvl:=E_LogSeverity.Debug, Msg:= F_Concat2(F_Concat2('gen grid point c:', TO_STRING(col)), F_Concat2('/r:', TO_STRING(row))));
      
      // - calculate x/y shift and rotation based on available CamPoints
      sTmpPoint.index := TO_DINT(col * _sDefGridSettings.nGridSizeY + row);
      sTmpPoint.x_ref := col * _sDefGridSettings.nGridPitchX;
      sTmpPoint.y_ref := row * _sDefGridSettings.nGridPitchY;
      sTmpPoint.dx    := dx;
      sTmpPoint.dy    := dy;
      sTmpPoint.col   := TO_DINT(col);
      sTmpPoint.row   := TO_DINT(row);
      sTmpPoint.valid := TRUE;
      storeDeformationPoint(sPoint:=sTmpPoint);    // save point to table
    END_FOR
    
    _nLocalGridColsGenerated := _nLocalGridColsGenerated + 1;
  END_IF
  
END_FOR


// set state variables which would be updated in PyUpdate/PyExed
_tExecutionTime := T#2MS;
_nErrorId := 0;
bPythonError := FALSE;
bPythonBusy := SEL(_nGridPoints >= _sDefGridSettings.nGridPoints, TRUE, FALSE); // all points generated
//bPythonBusy := SEL(_nGridCols   >= _sDefGridSettings.nGridSizeX,  TRUE, FALSE);  // all columns generated

fTrig_Done(CLK:=bPythonBusy);
IF fTrig_Done.Q THEN
  ;
END_IF

bPythonDeformationDone := NOT bPythonBusy;
END_METHOD

END_FUNCTION_BLOCK

// ---- POUs/Print/DefGrid/FB_PythonDeformation.TcPOU
FUNCTION_BLOCK FB_PythonDeformation EXTENDS FB_BasePrint
VAR
  // The variables below are accessed by the Python script. Do not change their names!
  // ------------------------------------------
  //FIFO Buffers
  fbFifoCamPoints : FB_DeformationPointFIFO; // Input FIFO, do not use Pop()
	fbFifoGridPoints : FB_DeformationPointFIFO; // Output FIFO, do not use Push()

	//Handshake variables
	fPythonPosition : LREAL := 0.0; (* Current position to process - should be kept constant while Python script is executing *)
	nPythonId : DINT := 0;   (* ct id for unique trace of ct in script *)
  
	bPythonStartUpdate : BOOL := FALSE; (* Tell the script to start its execution *)
	bPythonAbort : BOOL := FALSE; (* Abort any pending operation - NOT IMPLEMENTED *)
  
	bPythonBusy : BOOL := FALSE;
	bPythonUpdateDone : BOOL := FALSE; (* Set by the script when it's done or if error occurs *)
	bPythonError : BOOL := FALSE; (* Set by the script if any error occures during execution, cleared with abort - NOT IMPLEMENTED*)
  nPythonStatus : UDINT := 0; (*Set by the script status of deformation - NOT IMPLEMENTED*)
	bPythonDeformationDone : BOOL := FALSE; (* Set by the script when deformation if finished *)
  // ------------------------------------------
  
  // internal control
  _fbTimeout : TON; (* Counter with timeout *)
	_tExecutionTime : TIME := T#0S;   (*exection time local for scoping*)
  _bAborted : BOOL;
  
END_VAR

METHOD ExecPy : BOOL
VAR_OUTPUT
  bBusy : BOOL;
  nErrId : UDINT;
END_VAR
VAR
  _sTempPoint : ST_DeformationPoint;
END_VAR
// update FIFOs (external ADS access)
fbFifoCamPoints();
fbFifoGridPoints();

// work with script
IF bPythonBusy THEN // Pending job
	IF _fbTimeout.Q THEN // Timeout occurs
		_tExecutionTime := _fbTimeout.ET;
    bPythonAbort := TRUE;   // abort (pending operation) because id did not repond within timeout
		bPythonError := TRUE;   // set internal error
		nErrId := 1;
		bPythonBusy := FALSE;
    LogError(F_Concat4('Timeout during bPythonBusy, ExecTime:', TO_STRING(_tExecutionTime), ' Err:', TO_STRING(nErrId)));
	ELSIF bPythonUpdateDone THEN //Script done
		_tExecutionTime := _fbTimeout.ET;
		bPythonBusy := FALSE;
		IF bPythonError THEN
			nErrId := 2;
      LogError(F_Concat4('Error/abort requested by py, ExecTime:', TO_STRING(_tExecutionTime), ' Err:', TO_STRING(nErrId)));
		END_IF
  ELSIF _bAborted THEN      // abort if abort request set on ct
    bPythonBusy := FALSE;
    bPythonError := TRUE;   // set internal error
    nErrId := 3;
	END_IF
ELSIF bPythonAbort THEN
	bPythonStartUpdate := FALSE;
ELSE // Update/Job done  
  bPythonAbort := FALSE;
	bPythonStartUpdate := FALSE;
	bPythonUpdateDone := FALSE;
END_IF

_fbTimeout(IN := bPythonBusy);
END_METHOD

METHOD PROTECTED PopDeformationPoint :  BOOL;
VAR_OUTPUT
  sNewPoint : ST_DeformationPointAccurate;
END_VAR
VAR
  sPoint : ST_DeformationPoint;
END_VAR
IF fbFifoGridPoints.nCount > 0 THEN
  PopDeformationPoint := fbFifoGridPoints.Pop(sGridPoint=>sPoint);
  sNewPoint := F_DecodeDeformationPoint(sPoint:=sPoint, nResolution:=GVL_Deformation.nC_GridSubReso);
ELSE
  PopDeformationPoint := FALSE;
END_IF
END_METHOD

METHOD PROTECTED PushDeformationPoint : BOOL
VAR_INPUT
  sPoint : ST_DeformationPoint;
END_VAR
PushDeformationPoint:= fbFifoCamPoints.Push(sPoint);
END_METHOD

METHOD Reset
VAR_INPUT
END_VAR
fPythonPosition := 0.0;
//nPythonId := ;
bPythonStartUpdate := FALSE;
bPythonAbort := FALSE;
bPythonBusy := FALSE;
bPythonUpdateDone := FALSE;
bPythonError := FALSE;
nPythonStatus := 0;
bPythonDeformationDone := FALSE;

_fbTimeout(IN:=FALSE);
_bAborted := FALSE;

fbFifoCamPoints.Reset();
fbFifoGridPoints.Reset();
END_METHOD

METHOD UpdatePy : BOOL
VAR_INPUT
  fPosition : LREAL;
END_VAR
IF bPythonBusy THEN // Pending job
  UpdatePy:=FALSE;
  LogLvl(Lvl:=E_LogSeverity.Debug, Msg:='Python was still busy during updateDeformation');

ELSE // Job done

  IF NOT bPythonDeformationDone AND NOT bPythonAbort THEN // Sample input
    // start a update
    fPythonPosition := fPosition * GVL_Deformation.nC_GridSubReso;
    bPythonBusy := TRUE;
    bPythonError := FALSE;

    // Start script
    bPythonStartUpdate := TRUE;      
  END_IF

  UpdatePy:=TRUE;
END_IF
END_METHOD

END_FUNCTION_BLOCK

// ---- POUs/Print/DefGrid/FB_DeformationPointFIFO.TcPOU
FUNCTION_BLOCK FB_DeformationPointFIFO
VAR_OUTPUT
	nCount    : UINT;                 // Fill level
  nBufferSize : UINT := MAX_BUFFER_SIZE;
  nBufferItemSize : UINT := BUFFER_ITEM_SIZE;
END_VAR
VAR
	sBuffer 	: ARRAY[0..(MAX_BUFFER_SIZE-1)] OF ST_DeformationPoint;
	nHeadPtr  : UINT := 0;            // Point to the first non-empty idx
	nTailPtr  : UINT := 0;            // Pointer to the first free idx
  _bError    : BOOL;
END_VAR
VAR CONSTANT
	MAX_BUFFER_SIZE   : UINT := 1000;  // max. buffer size
	BUFFER_ITEM_SIZE  : UINT := SIZEOF(ST_DeformationPoint)/4; // Divide by 4 as we packed the ST_POINT with 32bits steps
END_VAR


(* now done async in method, this was dangerous...
// FIFO level
IF nTailPtr <= nHeadPtr THEN
	nCount := nHeadPtr - nTailPtr;
ELSE
	nCount := MAX_BUFFER_SIZE + nHeadPtr - nTailPtr;
END_IF
*)

PROPERTY bError : BOOL
GET
bError := _bError;
END_GET
END_PROPERTY

(*
  Get point from fifo queue. 
  :return: TRUE on success
*)
METHOD Pop : BOOL
VAR_OUTPUT
	sGridPoint : ST_DeformationPoint;
END_VAR
IF nCount = 0 THEN
  F_LogError('FB_DeformationPointFIFO is empty, cannot return an element');
  _bError := TRUE; 
  RETURN;
END_IF

sGridPoint := sBuffer[nTailPtr];
nTailPtr := (nTailPtr + 1) MOD MAX_BUFFER_SIZE;
nCount := nCount - 1;
_bError := FALSE;
Pop := TRUE;
END_METHOD

(*
  Add a new point to the fifo queue.
  :return: TRUE on success.
*)
METHOD Push : BOOL
VAR_INPUT
	sNewPoint : ST_DeformationPoint;
END_VAR
IF nCount >= MAX_BUFFER_SIZE THEN
  F_LogError('FB_DeformationPointFIFO overflow, element ignored');
  _bError := TRUE;
  RETURN;
END_IF

sBuffer[nHeadPtr] := sNewPoint;
nHeadPtr := (nHeadPtr + 1) MOD MAX_BUFFER_SIZE;
nCount := nCount + 1;
_bError := FALSE;
Push := TRUE;
END_METHOD

METHOD Reset : BOOL
VAR_INPUT
END_VAR
nTailPtr := 0;
nHeadPtr := 0;
nCount := 0;
_bError := 0;
END_METHOD

END_FUNCTION_BLOCK

// ---- POUs/Print/DefGrid/FB_CTManagerDefGrid.TcPOU
FUNCTION_BLOCK FB_CTManagerDefGrid EXTENDS FB_CTManager
VAR
  fbContainerInstances    : ARRAY[0..nC_MAX_CTS-1] OF FB_ContainerDefGrid;   // NOTE: 0 based array like base in library
  nCtr, nIndx : UDINT;
  _LogLevelCTs : E_LogSeverity := E_LogSeverity.Info;
END_VAR

// call CT manager base
SUPER^();

// call specific CT implementation
nCtr := 0;
WHILE nCtr < nListCount DO
  nIndx := ((nListTail + nCtr) MOD nC_MAX_CTS);    // calculate element index in list
  
  // cyclic call of CT body
  fbContainerInstances[nIndx]();
  
  nCtr := nCtr + 1;
END_WHILE

updateLogLevelsCTs();

(*
  Abort CTs
*)
METHOD AbortCts : BOOL
VAR_INPUT
  iCT : I_CT;     // reference CT 
  nSel : INT;     // selection: -1=all older (created before reference), 0=current only, 1=all newer (created after reference)
  Src : REFERENCE TO T_ErrSrc;
END_VAR
VAR
  iIterCt : I_CT;
  pCtSelected : POINTER TO FB_ContainerDefGrid;
END_VAR

// WARNING: This function is NOT tested!!! 
//    TODO: remove this comments when tested

IF nSel = 0 THEN
  // Abort referenced CT
  pCtSelected := GetContainerInstance(iCT:=iCT);
  IF pCtSelected <> 0 THEN
    pCtSelected^.AbortDeformation(sReason:=F_Concat2('CTM Abort CTs Sel=', TO_STRING(nSel)), Src:=Src, bHideLog:=FALSE);
  END_IF

